THIS^.testStartsWith(
	stringToTest := "",
	expectedString := ""
);
THIS^.testStartsWith(
	stringToTest := "not empty",
	expectedString := ""
);
THIS^.testStartsWith(
	stringToTest := "",
	expectedString := "not empty"
);
THIS^.testStartsWith(
	stringToTest := "not empty",
	expectedString := "not empty"
);
THIS^.testStartsWith(
	stringToTest := "{|}~",
	expectedString := "3649213469328"
);
THIS^.testStartsWith(
	stringToTest := "1one!",
	expectedString := "1"
);
THIS^.testStartsWith(
	stringToTest := "1one!",
	expectedString := "one"
);
THIS^.testStartsWith(
	stringToTest := "1one!",
	expectedString := "!"
);
THIS^.testStartsWith(
	stringToTest := "$0040$n$t$$$"$"",
	expectedString := "$n$t"
);
THIS^.testStartsWith(
	stringToTest := "$n$t$0040$$$"$"",
	expectedString := "$n$t"
);
THIS^.testStartsWith(
	stringToTest := "frontmiddleback",
	expectedString := "front"
);
THIS^.testStartsWith(
	stringToTest := "frontmiddleback",
	expectedString := "frontmiddlebackfront"
);
THIS^.testStartsWith(
	stringToTest := "backfrontmiddle",
	expectedString := "backmiddle"
);
THIS^.testStartsWith(
	stringToTest := "J;%_iTxQSk?6GfWewt}yMKh1)VXqPA@P1YQ:{EAg:8VJ,/FM;j)xJ[[AvYp/}}SzEgtfYS,1K0.5VtA+VJrB(p#55h2z##mw#F)Y@P6Jz9G@6vb=x#E!cYk(Svr@S*KiPJr1VZ6AjrNback4G=vBJd.E:=,k3!wmuGDe#ZKMD#Vx%?M_0&L0#vT]J,+)ZvU{w%8X0=:XzthmT0VG0QrwpXXCWpFxu6[b!c.BunYYfLQi.,?ut?-{jrC1phTHL)y",
	expectedString := "J;%_iTxQSk?6GfWewt}yMKh1)VXqPA@P1YQ:{EAg:8VJ,/FM;j)xJ[[AvYp/}}SzEgtfYS,1K0.5VtA+VJrB(p#55h2z##mw#F)Y@P6Jz9G@6vb=x#E!cYk(Svr@S*KiPJr1VZ6AjrNback4G=vBJd.E:=,k3!wmuGDe#ZKMD#Vx%?M_0&L0#vT]J,+)ZvU{w%8X0=:XzthmT0VG0QrwpXXCWpFxu6[b!c.BunYYfLQi.,?ut?-{jrC1phTHL)y"
);
THIS^.testStartsWith(
	stringToTest := "J;%_iTxQSk?6GfWewt}yMKh1)VXqPA@P1YQ:{EAg:8VJ,/FM;j)xJ[[AvYp/}}SzEgtfYS,1K0.5VtA+VJrB(p#55h2z##mw#F)Y@P6Jz9G@6vb=x#E!cYk(Svr@S*KiPJr1VZ6AjrNback4G=vBJd.E:=,k3!wmuGDe#ZKMD#Vx%?M_0&L0#vT]J,+)ZvU{w%8X0=:XzthmT0VG0QrwpXXCWpFxu6[b!c.BunYYfLQi.,?ut?-{jrC1phTHL)y",
	expectedString := "J;%_iTxQSk?6GfWewt}yMKh1)VXqPA@P1YQ:{EAg:8VJ,/FM;j)xJ[[AvYp/}}SzEgtfYS,1K0.5VtA+VJrB(p#55h2z##mw#F)Y@P6Jz9G@6vb=x#E!cYk(Svr@S*KiPJr1VZ6AjrNback4G=vBJd.E:=,k3!wmuGDe#ZKMD#Vx%?M_0&L0#vT]J,+)ZvU{w%8X0=:XzthmT0VG0QrwpXXCWpFxu6[b!c.BunYYfLQi.,?ut?-{jrC1phTHL)x"
);
THIS^.testStartsWith(
	stringToTest := "∮ E⋅da = Q,  n → ∞, ∑ f(i) = ∏ g(i), ∀x∈ℝ: ⌈x⌉ = −⌊−x⌋, α ∧ ¬β = ¬(¬α ∨ β)",
	expectedString := "∮ E⋅da = Q,  n → ∞"
);
THIS^.testStartsWith(
	stringToTest := "ℕ ⊆ ℕ₀ ⊂ ℤ ⊂ ℚ ⊂ ℝ ⊂ ℂ, ⊥ < a ≠ b ≡ c ≤ d ≪ ⊤ ⇒ (A ⇔ B), 2H₂ + O₂ ⇌ 2H₂O, R = 4.7 kΩ, ⌀ 200 mm",
	expectedString := "ℕ ⊆ ℕ₀ ⊂ ⊂ ℚ ⊂ ℝ ⊂ ℂ"
);
THIS^.testStartsWith(
	stringToTest := "ℕ ⊆ ℕ₀ ⊂ ℤ ⊂ ℚ ⊂ ℝ ⊂ ℂ, ⊥ < a ≠ b ≡ c ≤ d ≪ ⊤ ⇒ (A ⇔ B), 2H₂ + O₂ ⇌ 2H₂O, R = 4.7 kΩ, ⌀ 200 mm",
	expectedString := "ℕ ⊆ ℕ₀ ⊂ ℤ ⊂ ℚ ⊂ ℝ ⊂ ℂ, R = 4.7 kΩ, ⌀ 200 mm"
);
THIS^.testStartsWith(
	stringToTest := "ℕ ⊆ ℕ₀ ⊂ ℤ ⊂ ℚ ⊂ ℝ ⊂ ℂ, ⊥ < a ≠ b ≡ c ≤ d ≪ ⊤ ⇒ (A ⇔ B), 2H₂ + O₂ ⇌ 2H₂O, R = 4.7 kΩ, ⌀ 200 mm",
	expectedString := "ℕ ⊆ ℕ₀ ⊂ ℤ ⊂ ℚ ⊂ ℝ ⊂ ⊥"
);
THIS^.testStartsWith(
	stringToTest := "ði ıntəˈnæʃənəl fəˈnɛtık əsoʊsiˈeıʃn Y [ˈʏpsilɔn], Yen [jɛn], Yoga [ˈjoːgɑ]ˈnæʃənəl fəˈnɛtık ",
	expectedString := "ði ıntəˈnæʃənəl fəˈnɛtık"
);
THIS^.testStartsWith(
	stringToTest := "‚‘„“‘’“We’ve been here”´` †, ‡, ‰, •, 3–4, —, −5/+5, ™, …, 1lI|, 0OD, 8B, €",
	expectedString := "‚‘„“‘’“We’ve been here”´` †, ‡, ‰, •, 3–4, —, −5/+5, ™, …, 1lI|, 0OD, 8B, €"
);
THIS^.testStartsWith(
	stringToTest := "Σὲ γνωρίζω ἀπὸ τὴν κόψη τοῦ σπαθιοῦ τὴν τρομερή,",
	expectedString := "τὴν κόψη τοῦ σπαθ"
);
THIS^.testStartsWith(
	stringToTest := "გთხოვთ ახლავე გაიაროთ რეგისტრაცია Unicode-ის მეათე საერთაშორისო კონფერენციაზე დასასწრებად, რომელიც გაიმართება",
	expectedString := "გთხოვთ ახლავე გაიაროთ რეგისტრაცია"
);
THIS^.testStartsWith(
	stringToTest := "Зарегистрируйтесь сейчас на Десятую Международную Конференцию по Unicode, которая состоится 10-12 марта 1997 года в",
	expectedString := "Международную Конференцию по Unicode, которая"
);
THIS^.testStartsWith(
	stringToTest := "๏ แผ่นดินฮั่นเสื่อมโทรมแสนสังเวช  พระปกเกศกองบู๊กู้ขึ้นใหม่
  สิบสองกษัตริย์ก่อนหน้าแลถัดไป       สององค์ไซร้โง่เขลาเบาปัญญา ",
	expectedString := "๏ แผ่นดินฮั่นเสื่อมโทรมแสนสังเวช " 
);
THIS^.testStartsWith(
	stringToTest := " ሰማይ አይታረስ ንጉሥ አይከሰስ። ብላ ካለኝ እንደአባቴ በቆመጠኝ።",
	expectedString := "አይታረስ ንጉሥ አይከሰስ። በቆመጠኝ።"
);
THIS^.testStartsWith(
	stringToTest := " ᚻᛖ ᚳᚹᚫᚦ ᚦᚫᛏ ᚻᛖ ᛒᚢᛞᛖ ᚩᚾ ᚦᚫᛗ ᛚᚪᚾᛞᛖ ᚾᚩᚱᚦᚹᛖᚪᚱᛞᚢᛗ ᚹᛁᚦ ᚦᚪ ᚹᛖᛥᚫ",
	expectedString := " ᚻᛖ ᚳᚹᚫᚦ ᚦᚫᛏ ᚻᛖ"
);
THIS^.testStartsWith(
	stringToTest := "⡍⠔⠙⠖ ⡊ ⠙⠕⠝⠰⠞ ⠍⠑⠁⠝ ⠞⠕ ⠎⠁⠹ ⠹⠁⠞ ⡊ ⠅⠝⠪⠂ ⠕⠋ ⠍⠹
  ⠪⠝ ⠅⠝⠪⠇⠫⠛⠑⠂ ⠱⠁⠞ ⠹⠻⠑ ⠊⠎ ⠏⠜⠞⠊⠊⠥⠇⠜⠇⠹ ⠙⠑⠁⠙ ⠁⠃⠳⠞",
	expectedString := "⠱⠁⠞ ⠹⠻⠑ ⠊⠎ ⠏⠜⠞⠊⠊⠥⠇⠜⠇⠹ ⠙"
);
THIS^.testStartsWith(
	stringToTest := "╔══╦══╗  ┌──┬──┐  ╭──┬──╮  ╭──┬──╮  ┏━━┳━━┓  ┎┒┏┑   ╷  ╻ ┏┯┓ ┌┰┐    ▊ ╱╲╱╲╳╳╳",
	expectedString := "╔══╦══╗  ┌──┬──┐"
);

THIS^.testStartsWithIgnoreCase(
	stringToTest := "UPPERCASE",
	expectedString := "UPPER"
);
THIS^.testStartsWithIgnoreCase(
	stringToTest := "lowercase",
	expectedString := "lower"
);
THIS^.testStartsWithIgnoreCase(
	stringToTest := "UPPERCASE",
	expectedString := "upper"
);
THIS^.testStartsWithIgnoreCase(
	stringToTest := "lowercase",
	expectedString := "LOWER"
);
THIS^.testStartsWithIgnoreCase(
	stringToTest := "lower",
	expectedString := "UPPER"
);
THIS^.testStartsWithIgnoreCase(
	stringToTest := "⌷←⍳→⍴∆∇⊃‾⍎⍕⌈UPPERCASE",
	expectedString := "⌷←⍳→⍴∆∇⊃‾⍎⍕⌈upper"
);
THIS^.testStartsWithIgnoreCase(
	stringToTest := "⌷←⍳→⍴∆∇⊃‾⍎⍕⌈UPPERCASE",
	expectedString := "⌷←⍳→⍴∆∇⊃‾⍎⍕⌈|upper"
);

THIS^.testStartsWithTrim(
	stringToTest := "$tfrontmiddleback",
	expectedString := "front"
);
THIS^.testStartsWithTrim(
	stringToTest := "frontmiddleback",
	expectedString := "$tfront"
);
THIS^.testStartsWithTrim(
	stringToTest := "$0020frontmiddleback",
	expectedString := "front"
);
THIS^.testStartsWithTrim(
	stringToTest := "frontmiddleback",
	expectedString := "$0020front"
);
THIS^.testStartsWithTrim(
	stringToTest := "$t$n$r$p$lfrontmiddleback",
	expectedString := "$0020$r$t$n$l$pfront"
);
THIS^.testStartsWithTrim(
	stringToTest := "$t$n$r$p$lfrontmiddleback",
	expectedString := "$0020$t$n$r$p$lfront"
);
THIS^.testStartsWithTrim(
	stringToTest := "$t$n$r$p$l⌷←⍳→⍴∆∇⊃‾⍎⍕⌈frontmiddleback$t$n$r$p$l",
	expectedString := "⌷←⍳→⍴∆∇⊃‾⍎⍕⌈front"
);
THIS^.testStartsWithTrim(
	stringToTest := "$t$n$r$p$l⌷←⍳→⍴∆∇⊃‾⍎⍕⌈frontmiddleback$t$n$r$p$l",
	expectedString := "⌷←⍳→⍴∆∇⊃‾⍎⍕front⌈"
);

TcUnit.TEST_FINISHED();
END_METHOD

(*
short summary
==================
This test method tests ``assert.string.unicode.contains``
method of CNM_AssertionInterfaces library with various inputs

.. <legal notes>

legal notes
=================
| SPDX-FileCopyrightText: © 2022 ekvip automation GmbH <info@ekvip.de>
| SPDX-License-Identifier: Apache-2.0
| For details check: Apache-2.0_

.. _Apache-2.0: https://www.apache.org/licenses/LICENSE-2.0

.. </legal notes>

*)


METHOD testContains : BOOL
VAR_INPUT
	(* for the test it's the parameter ``stringToCheck`` *)
	stringToTest 					:WSTRING(Tc2_System.MAX_STRING_LENGTH);
	(* for the test it's the parameter ``searchString`` *)
	expectedString					:WSTRING(Tc2_System.MAX_STRING_LENGTH);
END_VAR
VAR 
	(* just the expectation if the assertion to test must be worng or true *)
	assertionIsWrong				:BOOL;
	(* contains the format string for the test message *)
	message							:Tc2_System.T_MaxString;
	(* used for placeholder string if stringToTest can't be printed *)
	stringToTestAsString 			:Tc2_System.T_MaxString;
	(* used for placeholder string if expectedString can't be printed *)
	expectedStringAsString 			:Tc2_System.T_MaxString;
	(* contains stringToTest in normalized form *)
	normalizedStringToTest			:WSTRING(Tc2_System.MAX_STRING_LENGTH);
	(* contains expectedString in normalized form *)
	normalizedExpectedString		:WSTRING(Tc2_System.MAX_STRING_LENGTH);
	(* holds characterCount of ``expectedString`` *)
	expectedCharacterCount			:UDINT;
	(* TwinCAT printf with the test message *)
	messageStringBuilder			:Tc2_Utilities.FB_FormatString;
	(* hold stringToCheck before assertion *)
	stringToTestBeforeAssertion		:WSTRING(Tc2_System.MAX_STRING_LENGTH);
	(* hold stringToCheck before assertion *)
	expectedStringBeforeAssertion	:WSTRING(Tc2_System.MAX_STRING_LENGTH);
END_VAR
THIS^.assertorContainer.resetAssertor();

stringToTestBeforeAssertion := stringToTest;
expectedStringBeforeAssertion := expectedString;

CNM_UnicodeUtilities.GetUtf16StringLength(
	utf16StringAddress := ADR(expectedString),
	characterCount => expectedCharacterCount
);
assertionIsWrong := ((
		CNM_UnicodeUtilities.FindInUtf16String(
			ADR(stringToTest),
			ADR(expectedString),
		) = 0
	) AND (
		expectedCharacterCount <> 0
	)
);

message := SEL(
	assertionIsWrong,
	'stringToCheck is $'%s$' searchString is $'%s$' assertion must be TRUE', 
	'stringToCheck is $'%s$' searchString is $'%s$' assertion must be FALSE'
);
Tc2_Utilities.WSTRING_TO_STRING2(ADR(stringToTestAsString), ADR(stringToTest), SIZEOF(stringToTestAsString));
Tc2_Utilities.WSTRING_TO_STRING2(ADR(expectedStringAsString), ADR(expectedString), SIZEOF(expectedStringAsString));

IF (
		Tc2_Standard.WLEN(stringToTest) = TO_UINT(Tc2_System.MAX_STRING_LENGTH)
) THEN
	stringToTestAsString := 'String with Tc2_System.MAX_STRING_LENGTH characters';
END_IF
IF (
		Tc2_Standard.WLEN(expectedString) = TO_UINT(Tc2_System.MAX_STRING_LENGTH)
) THEN
	expectedStringAsString := 'String with Tc2_System.MAX_STRING_LENGTH characters';
END_IF

messageStringBuilder(
	sFormat := message,
	arg1 := THIS^.AnyToArg(stringToTestAsString),
	arg2 := THIS^.AnyToArg(expectedStringAsString)
);

THIS^.assertorContainer.assertor.assert.strings.unicode.contains(
	stringToCheck := stringToTest,
	searchString := expectedString,
	ignoreCases := FALSE,
	normalizeStrings := FALSE,
	message			:= ''
);

THIS^.AssertEquals_BOOL(
	Expected 	:= assertionIsWrong,
	Actual 		:= THIS^.assertorContainer.wasAssertionWrong,
	Message 	:= messageStringBuilder.sOut
);

THIS^.AssertEquals_WSTRING(
	Expected 	:= stringToTestBeforeAssertion,
	Actual 		:= stringToTest,
	Message 	:= 'the assertion changed $'stringToTest$''
);

THIS^.AssertEquals_WSTRING(
	Expected 	:= expectedStringBeforeAssertion,
	Actual 		:= expectedString,
	Message 	:= 'the assertion changed $'expectedString$''
);

THIS^.assertorContainer.resetAssertor();

CNM_UnicodeUtilities.NormalizeUtf16String(
	utf16StringBuffer := ADR(stringToTest),
	bufferSize := Tc2_System.MAX_STRING_LENGTH * 2 + 2,
	normalizedStringBuffer := ADR(normalizedStringToTest),
	normalForm := CNM_UnicodeUtilities.NormalizationForm.NFD
);
CNM_UnicodeUtilities.NormalizeUtf16String(
	utf16StringBuffer := ADR(expectedString),
	bufferSize := Tc2_System.MAX_STRING_LENGTH * 2 + 2,
	normalizedStringBuffer := ADR(normalizedExpectedString),
	normalForm := CNM_UnicodeUtilities.NormalizationForm.NFD
);

CNM_UnicodeUtilities.GetUtf16StringLength(
	utf16StringAddress := ADR(normalizedExpectedString),
	characterCount => expectedCharacterCount
);
assertionIsWrong := ((
		CNM_UnicodeUtilities.FindInUtf16String(
			ADR(normalizedStringToTest),
			ADR(normalizedExpectedString),
		) = 0
	) AND (
		expectedCharacterCount <> 0
	)
);

THIS^.assertorContainer.assertor.assert.strings.unicode.contains(
	stringToCheck := stringToTest,
	searchString := expectedString,
	ignoreCases := FALSE,
	normalizeStrings := TRUE,
	message			:= ''
);

THIS^.AssertEquals_BOOL(
	Expected 	:= assertionIsWrong,
	Actual 		:= THIS^.assertorContainer.wasAssertionWrong,
	Message 	:= messageStringBuilder.sOut
);

THIS^.AssertEquals_WSTRING(
	Expected 	:= stringToTestBeforeAssertion,
	Actual 		:= stringToTest,
	Message 	:= 'the assertion changed $'stringToTest$''
);

THIS^.AssertEquals_WSTRING(
	Expected 	:= expectedStringBeforeAssertion,
	Actual 		:= expectedString,
	Message 	:= 'the assertion changed $'expectedString$''
);
END_METHOD

(*
short summary
==================
This test method tests ``assert.string.unicode.contains``
method of CNM_AssertionInterfaces library with various inputs

.. <legal notes>

legal notes
=================
| SPDX-FileCopyrightText: © 2022 ekvip automation GmbH <info@ekvip.de>
| SPDX-License-Identifier: Apache-2.0
| For details check: Apache-2.0_

.. _Apache-2.0: https://www.apache.org/licenses/LICENSE-2.0

.. </legal notes>

*)


METHOD testContainsIgnoreCase : BOOL
VAR_INPUT
	(* for the test it's the parameter ``stringToCheck`` *)
	stringToTest  	:WSTRING(Tc2_System.MAX_STRING_LENGTH);
	(* for the test it's the parameter ``searchString`` *)
	expectedString	:WSTRING(Tc2_System.MAX_STRING_LENGTH);
END_VAR
VAR 
	(* just the expectation if the assertion to test must be worng or true *)
	assertionIsWrong				:BOOL;
	(* contains the format string for the test message *)
	message							:Tc2_System.T_MaxString;
	(* contains ´´stringToTest´´ in upper case *)
	upperStringToTest				:WSTRING(Tc2_System.MAX_STRING_LENGTH);
	(* contains ´´expectedString´´ in upper case *)
	upperExpectedString				:WSTRING(Tc2_System.MAX_STRING_LENGTH);
	(* used for placeholder string if stringToTest can't be printed *)
	stringToTestAsString 			:Tc2_System.T_MaxString;
	(* used for placeholder string if expectedString can't be printed *)
	expectedStringAsString			:Tc2_System.T_MaxString;
	(* contains stringToTest in normalized form *)
	normalizedStringToTest			:WSTRING(Tc2_System.MAX_STRING_LENGTH);
	(* contains expectedString in normalized form *)
	normalizedExpectedString		:WSTRING(Tc2_System.MAX_STRING_LENGTH);
	(* contains stringToTest in normalized form in upper case*)
	normalizedUpperStringToTest		:WSTRING(Tc2_System.MAX_STRING_LENGTH);
	(* contains expectedString in normalized form in upper case*)
	normalizedUpperExpectedString	:WSTRING(Tc2_System.MAX_STRING_LENGTH);
	(* holds characterCount of ``expectedString`` *)
	expectedCharacterCount			:UDINT;
	(* TwinCAT printf with the test message *)
	messageStringBuilder			:Tc2_Utilities.FB_FormatString;
	(* hold stringToCheck before assertion *)
	stringToTestBeforeAssertion		:WSTRING(Tc2_System.MAX_STRING_LENGTH);
	(* hold stringToCheck before assertion *)
	expectedStringBeforeAssertion	:WSTRING(Tc2_System.MAX_STRING_LENGTH);
END_VAR
THIS^.assertorContainer.resetAssertor();

stringToTestBeforeAssertion := stringToTest;
expectedStringBeforeAssertion := expectedString;

upperStringToTest := stringToTest;
upperExpectedString := expectedString;

// both Strings to upper case
CNM_UnicodeUtilities.GetUpperCaseUtf16(ADR(upperStringToTest));
CNM_UnicodeUtilities.GetUpperCaseUtf16(ADR(upperExpectedString));

CNM_UnicodeUtilities.GetUtf16StringLength(
	utf16StringAddress := ADR(upperExpectedString),
	characterCount => expectedCharacterCount
);
assertionIsWrong := ((
		CNM_UnicodeUtilities.FindInUtf16String(
			ADR(upperStringToTest),
			ADR(upperExpectedString),
		) = 0
	) AND (
		expectedCharacterCount <> 0
	)
);

message := SEL(
	assertionIsWrong,
	'stringToCheck is $'%s$' searchString is $'%s$' assertion must be TRUE', 
	'stringToCheck is $'%s$' searchString is $'%s$' assertion must be FALSE'
);

Tc2_Utilities.WSTRING_TO_STRING2(ADR(stringToTestAsString), ADR(stringToTest), SIZEOF(stringToTestAsString));
Tc2_Utilities.WSTRING_TO_STRING2(ADR(expectedStringAsString), ADR(expectedString), SIZEOF(expectedStringAsString));

IF (
		Tc2_Standard.WLEN(stringToTest) = TO_UINT(Tc2_System.MAX_STRING_LENGTH)
) THEN
	stringToTestAsString := 'String with Tc2_System.MAX_STRING_LENGTH characters';
END_IF
IF (
		Tc2_Standard.WLEN(expectedString) = TO_UINT(Tc2_System.MAX_STRING_LENGTH)
) THEN
	expectedStringAsString := 'String with Tc2_System.MAX_STRING_LENGTH characters';
END_IF

messageStringBuilder(
	sFormat := message,
	arg1 := THIS^.AnyToArg(stringToTestAsString),
	arg2 := THIS^.AnyToArg(expectedStringAsString)
);


THIS^.assertorContainer.assertor.assert.strings.unicode.contains(
	stringToCheck := stringToTest,
	searchString := expectedString,
	ignoreCases := TRUE,
	normalizeStrings := FALSE,
	message			:= ''
);

THIS^.AssertEquals_BOOL(
	Expected 	:= assertionIsWrong,
	Actual 		:= THIS^.assertorContainer.wasAssertionWrong,
	Message 	:= messageStringBuilder.sOut
);

THIS^.AssertEquals_WSTRING(
	Expected 	:= stringToTestBeforeAssertion,
	Actual 		:= stringToTest,
	Message 	:= 'the assertion changed $'stringToTest$''
);

THIS^.AssertEquals_WSTRING(
	Expected 	:= expectedStringBeforeAssertion,
	Actual 		:= expectedString,
	Message 	:= 'the assertion changed $'expectedString$''
);

THIS^.assertorContainer.resetAssertor();

CNM_UnicodeUtilities.NormalizeUtf16String(
	utf16StringBuffer := ADR(stringToTest),
	bufferSize := Tc2_System.MAX_STRING_LENGTH * 2 + 2,
	normalizedStringBuffer := ADR(normalizedStringToTest),
	normalForm := CNM_UnicodeUtilities.NormalizationForm.NFD
);
CNM_UnicodeUtilities.NormalizeUtf16String(
	utf16StringBuffer := ADR(expectedString),
	bufferSize := Tc2_System.MAX_STRING_LENGTH * 2 + 2,
	normalizedStringBuffer := ADR(normalizedExpectedString),
	normalForm := CNM_UnicodeUtilities.NormalizationForm.NFD
);

normalizedUpperStringToTest := normalizedStringToTest;
normalizedUpperExpectedString := normalizedExpectedString;
CNM_UnicodeUtilities.GetUpperCaseUtf16(ADR(normalizedUpperStringToTest));
CNM_UnicodeUtilities.GetUpperCaseUtf16(ADR(normalizedUpperExpectedString));


CNM_UnicodeUtilities.GetUtf16StringLength(
	utf16StringAddress := ADR(normalizedUpperExpectedString),
	characterCount => expectedCharacterCount
);
assertionIsWrong := ((
		CNM_UnicodeUtilities.FindInUtf16String(
			ADR(normalizedUpperStringToTest),
			ADR(normalizedUpperExpectedString),
		) = 0
	) AND (
		expectedCharacterCount <> 0
	)
);

THIS^.assertorContainer.assertor.assert.strings.unicode.contains(
	stringToCheck := stringToTest,
	searchString := expectedString,
	ignoreCases := TRUE,
	normalizeStrings := TRUE,
	message			:= ''
);

THIS^.AssertEquals_BOOL(
	Expected 	:= assertionIsWrong,
	Actual 		:= THIS^.assertorContainer.wasAssertionWrong,
	Message 	:= messageStringBuilder.sOut
);

THIS^.AssertEquals_WSTRING(
	Expected 	:= stringToTestBeforeAssertion,
	Actual 		:= stringToTest,
	Message 	:= 'the assertion changed $'stringToTest$''
);

THIS^.AssertEquals_WSTRING(
	Expected 	:= expectedStringBeforeAssertion,
	Actual 		:= expectedString,
	Message 	:= 'the assertion changed $'expectedString$''
);
END_METHOD

(*
short summary
==================
This test method tests ``assert.string.unicode.containsNo``
method of CNM_AssertionInterfaces library with various inputs

.. <legal notes>

legal notes
=================
| SPDX-FileCopyrightText: © 2022 ekvip automation GmbH <info@ekvip.de>
| SPDX-License-Identifier: Apache-2.0
| For details check: Apache-2.0_

.. _Apache-2.0: https://www.apache.org/licenses/LICENSE-2.0

.. </legal notes>

*)


METHOD testContainsNo : BOOL
VAR_INPUT
	(* for the test it's the parameter ``stringToCheck`` *)
	stringToTest  			:WSTRING(Tc2_System.MAX_STRING_LENGTH);
	(* for the test it's the parameter ``searchString`` *)
	expectedString			:WSTRING(Tc2_System.MAX_STRING_LENGTH);
END_VAR
VAR 
	(* just the expectation if the assertion to test must be worng or true *)
	assertionIsWrong				:BOOL;
	(* contains the format string for the test message *)
	message							:Tc2_System.T_MaxString;
	(* used for placeholder string if stringToTest can't be printed *)
	stringToTestAsString 			:Tc2_System.T_MaxString;
	(* used for placeholder string if expectedString can't be printed *)
	expectedStringAsString 			:Tc2_System.T_MaxString;
	(* contains stringToTest in normalized form *)
	normalizedStringToTest			:WSTRING(Tc2_System.MAX_STRING_LENGTH);
	(* contains expectedString in normalized form *)
	normalizedExpectedString		:WSTRING(Tc2_System.MAX_STRING_LENGTH);
	(* holds characterCount of ``expectedString`` *)
	expectedCharacterCount			:UDINT;
	(* TwinCAT printf with the test message *)
	messageStringBuilder			:Tc2_Utilities.FB_FormatString;
	(* hold stringToCheck before assertion *)
	stringToTestBeforeAssertion		:WSTRING(Tc2_System.MAX_STRING_LENGTH);
	(* hold stringToCheck before assertion *)
	expectedStringBeforeAssertion	:WSTRING(Tc2_System.MAX_STRING_LENGTH);
END_VAR
THIS^.assertorContainer.resetAssertor();

stringToTestBeforeAssertion := stringToTest;
expectedStringBeforeAssertion := expectedString;

CNM_UnicodeUtilities.GetUtf16StringLength(
	utf16StringAddress := ADR(expectedString),
	characterCount => expectedCharacterCount
);
assertionIsWrong := ((
		CNM_UnicodeUtilities.FindInUtf16String(
			ADR(stringToTest),
			ADR(expectedString),
		) > 0
	) OR (
		expectedCharacterCount = 0
	)
);

message := SEL(
	assertionIsWrong,
	'stringToCheck is $'%s$' searchString is $'%s$' assertion must be TRUE', 
	'stringToCheck is $'%s$' searchString is $'%s$' assertion must be FALSE'
);

Tc2_Utilities.WSTRING_TO_STRING2(ADR(stringToTestAsString), ADR(stringToTest), SIZEOF(stringToTestAsString));
Tc2_Utilities.WSTRING_TO_STRING2(ADR(expectedStringAsString), ADR(expectedString), SIZEOF(expectedStringAsString));

IF (
		Tc2_Standard.WLEN(stringToTest) = TO_UINT(Tc2_System.MAX_STRING_LENGTH)
) THEN
	stringToTestAsString := 'String with Tc2_System.MAX_STRING_LENGTH characters';
END_IF
IF (
		Tc2_Standard.WLEN(expectedString) = TO_UINT(Tc2_System.MAX_STRING_LENGTH)
) THEN
	expectedStringAsString := 'String with Tc2_System.MAX_STRING_LENGTH characters';
END_IF

messageStringBuilder(
	sFormat := message,
	arg1 := THIS^.AnyToArg(stringToTestAsString),
	arg2 := THIS^.AnyToArg(expectedStringAsString)
);


THIS^.assertorContainer.assertor.assert.strings.unicode.containsNo(
	stringToCheck := stringToTest,
	searchString := expectedString,
	ignoreCases := FALSE,
	normalizeStrings := FALSE,
	message			:= ''
);

THIS^.AssertEquals_BOOL(
	Expected 	:= assertionIsWrong,
	Actual 		:= THIS^.assertorContainer.wasAssertionWrong,
	Message 	:= messageStringBuilder.sOut
);

THIS^.AssertEquals_WSTRING(
	Expected 	:= stringToTestBeforeAssertion,
	Actual 		:= stringToTest,
	Message 	:= 'the assertion changed $'stringToTest$''
);

THIS^.AssertEquals_WSTRING(
	Expected 	:= expectedStringBeforeAssertion,
	Actual 		:= expectedString,
	Message 	:= 'the assertion changed $'expectedString$''
);

THIS^.assertorContainer.resetAssertor();

CNM_UnicodeUtilities.NormalizeUtf16String(
	utf16StringBuffer := ADR(stringToTest),
	bufferSize := Tc2_System.MAX_STRING_LENGTH * 2 + 2,
	normalizedStringBuffer := ADR(normalizedStringToTest),
	normalForm := CNM_UnicodeUtilities.NormalizationForm.NFD
);
CNM_UnicodeUtilities.NormalizeUtf16String(
	utf16StringBuffer := ADR(expectedString),
	bufferSize := Tc2_System.MAX_STRING_LENGTH * 2 + 2,
	normalizedStringBuffer := ADR(normalizedExpectedString),
	normalForm := CNM_UnicodeUtilities.NormalizationForm.NFD
);

CNM_UnicodeUtilities.GetUtf16StringLength(
	utf16StringAddress := ADR(normalizedExpectedString),
	characterCount => expectedCharacterCount
);
assertionIsWrong := ((
		CNM_UnicodeUtilities.FindInUtf16String(
			ADR(normalizedStringToTest),
			ADR(normalizedExpectedString),
		) > 0
	) OR (
		expectedCharacterCount = 0
	)
);

THIS^.assertorContainer.assertor.assert.strings.unicode.containsNo(
	stringToCheck := stringToTest,
	searchString := expectedString,
	ignoreCases := FALSE,
	normalizeStrings := TRUE,
	message			:= ''
);

THIS^.AssertEquals_BOOL(
	Expected 	:= assertionIsWrong,
	Actual 		:= THIS^.assertorContainer.wasAssertionWrong,
	Message 	:= messageStringBuilder.sOut
);

THIS^.AssertEquals_WSTRING(
	Expected 	:= stringToTestBeforeAssertion,
	Actual 		:= stringToTest,
	Message 	:= 'the assertion changed $'stringToTest$''
);

THIS^.AssertEquals_WSTRING(
	Expected 	:= expectedStringBeforeAssertion,
	Actual 		:= expectedString,
	Message 	:= 'the assertion changed $'expectedString$''
);
END_METHOD

(*
short summary
==================
This test method tests ``assert.string.unicode.containsNo``
method of CNM_AssertionInterfaces library with various inputs

.. <legal notes>

legal notes
=================
| SPDX-FileCopyrightText: © 2022 ekvip automation GmbH <info@ekvip.de>
| SPDX-License-Identifier: Apache-2.0
| For details check: Apache-2.0_

.. _Apache-2.0: https://www.apache.org/licenses/LICENSE-2.0

.. </legal notes>

*)


METHOD testContainsNoIgnoreCase : BOOL
VAR_INPUT
	(* for the test it's the parameter ``stringToCheck`` *)
	stringToTest  	:WSTRING(Tc2_System.MAX_STRING_LENGTH);
	(* for the test it's the parameter ``searchString`` *)
	expectedString	:WSTRING(Tc2_System.MAX_STRING_LENGTH);
END_VAR
VAR 
	(* just the expectation if the assertion to test must be worng or true *)
	assertionIsWrong				:BOOL;
	(* contains the format string for the test message *)
	message							:Tc2_System.T_MaxString;
	(* contains ´´stringToTest´´ in upper case *)
	upperStringToTest				:WSTRING(Tc2_System.MAX_STRING_LENGTH);
	(* contains ´´expectedString´´ in upper case *)
	upperExpectedString				:WSTRING(Tc2_System.MAX_STRING_LENGTH);
	(* used for placeholder string if stringToTest can't be printed *)
	stringToTestAsString 			:Tc2_System.T_MaxString;
	(* used for placeholder string if expectedString can't be printed *)
	expectedStringAsString 			:Tc2_System.T_MaxString;
	(* contains stringToTest in normalized form *)
	normalizedStringToTest			:WSTRING(Tc2_System.MAX_STRING_LENGTH);
	(* contains expectedString in normalized form *)
	normalizedExpectedString		:WSTRING(Tc2_System.MAX_STRING_LENGTH);
	(* contains stringToTest in normalized form in upper case*)
	normalizedUpperStringToTest		:WSTRING(Tc2_System.MAX_STRING_LENGTH);
	(* contains expectedString in normalized form in upper case*)
	normalizedUpperExpectedString	:WSTRING(Tc2_System.MAX_STRING_LENGTH);
	(* holds characterCount of ``expectedString`` *)
	expectedCharacterCount			:UDINT;
	(* TwinCAT printf with the test message *)
	messageStringBuilder			:Tc2_Utilities.FB_FormatString;
	(* hold stringToCheck before assertion *)
	stringToTestBeforeAssertion		:WSTRING(Tc2_System.MAX_STRING_LENGTH);
	(* hold stringToCheck before assertion *)
	expectedStringBeforeAssertion	:WSTRING(Tc2_System.MAX_STRING_LENGTH);
END_VAR
THIS^.assertorContainer.resetAssertor();

stringToTestBeforeAssertion := stringToTest;
expectedStringBeforeAssertion := expectedString;

upperStringToTest := stringToTest;
upperExpectedString := expectedString;

// both Strings to upper case
CNM_UnicodeUtilities.GetUpperCaseUtf16(ADR(upperStringToTest));
CNM_UnicodeUtilities.GetUpperCaseUtf16(ADR(upperExpectedString));

CNM_UnicodeUtilities.GetUtf16StringLength(
	utf16StringAddress := ADR(upperExpectedString),
	characterCount => expectedCharacterCount
);
assertionIsWrong := ((
		CNM_UnicodeUtilities.FindInUtf16String(
			ADR(upperStringToTest),
			ADR(upperExpectedString),
		) > 0
	) OR (
		expectedCharacterCount = 0
	)
);

message := SEL(
	assertionIsWrong,
	'stringToCheck is $'%s$' searchString is $'%s$' assertion must be TRUE', 
	'stringToCheck is $'%s$' searchString is $'%s$' assertion must be FALSE'
);

Tc2_Utilities.WSTRING_TO_STRING2(ADR(stringToTestAsString), ADR(stringToTest), SIZEOF(stringToTestAsString));
Tc2_Utilities.WSTRING_TO_STRING2(ADR(expectedStringAsString), ADR(expectedString), SIZEOF(expectedStringAsString));

IF (
		Tc2_Standard.WLEN(stringToTest) = TO_UINT(Tc2_System.MAX_STRING_LENGTH)
) THEN
	stringToTestAsString := 'String with Tc2_System.MAX_STRING_LENGTH characters';
END_IF
IF (
		Tc2_Standard.WLEN(expectedString) = TO_UINT(Tc2_System.MAX_STRING_LENGTH)
) THEN
	expectedStringAsString := 'String with Tc2_System.MAX_STRING_LENGTH characters';
END_IF

messageStringBuilder(
	sFormat := message,
	arg1 := THIS^.AnyToArg(stringToTestAsString),
	arg2 := THIS^.AnyToArg(expectedStringAsString)
);


THIS^.assertorContainer.assertor.assert.strings.unicode.containsNo(
	stringToCheck := stringToTest,
	searchString := expectedString,
	ignoreCases := TRUE,
	normalizeStrings := FALSE,
	message			:= ''
);

THIS^.AssertEquals_BOOL(
	Expected 	:= assertionIsWrong,
	Actual 		:= THIS^.assertorContainer.wasAssertionWrong,
	Message 	:= messageStringBuilder.sOut
);

THIS^.AssertEquals_WSTRING(
	Expected 	:= stringToTestBeforeAssertion,
	Actual 		:= stringToTest,
	Message 	:= 'the assertion changed $'stringToTest$''
);

THIS^.AssertEquals_WSTRING(
	Expected 	:= expectedStringBeforeAssertion,
	Actual 		:= expectedString,
	Message 	:= 'the assertion changed $'expectedString$''
);

THIS^.assertorContainer.resetAssertor();

CNM_UnicodeUtilities.NormalizeUtf16String(
	utf16StringBuffer := ADR(stringToTest),
	bufferSize := Tc2_System.MAX_STRING_LENGTH * 2 + 2,
	normalizedStringBuffer := ADR(normalizedStringToTest),
	normalForm := CNM_UnicodeUtilities.NormalizationForm.NFD
);
CNM_UnicodeUtilities.NormalizeUtf16String(
	utf16StringBuffer := ADR(expectedString),
	bufferSize := Tc2_System.MAX_STRING_LENGTH * 2 + 2,
	normalizedStringBuffer := ADR(normalizedExpectedString),
	normalForm := CNM_UnicodeUtilities.NormalizationForm.NFD
);

normalizedUpperStringToTest := normalizedStringToTest;
normalizedUpperExpectedString := normalizedExpectedString;
CNM_UnicodeUtilities.GetUpperCaseUtf16(ADR(normalizedUpperStringToTest));
CNM_UnicodeUtilities.GetUpperCaseUtf16(ADR(normalizedUpperExpectedString));


CNM_UnicodeUtilities.GetUtf16StringLength(
	utf16StringAddress := ADR(normalizedUpperExpectedString),
	characterCount => expectedCharacterCount
);
assertionIsWrong := ((
		CNM_UnicodeUtilities.FindInUtf16String(
			ADR(normalizedUpperStringToTest),
			ADR(normalizedUpperExpectedString),
		) > 0
	) OR (
		expectedCharacterCount = 0
	)
);

THIS^.assertorContainer.assertor.assert.strings.unicode.containsNo(
	stringToCheck := stringToTest,
	searchString := expectedString,
	ignoreCases := TRUE,
	normalizeStrings := TRUE,
	message			:= ''
);

THIS^.AssertEquals_BOOL(
	Expected 	:= assertionIsWrong,
	Actual 		:= THIS^.assertorContainer.wasAssertionWrong,
	Message 	:= messageStringBuilder.sOut
);

THIS^.AssertEquals_WSTRING(
	Expected 	:= stringToTestBeforeAssertion,
	Actual 		:= stringToTest,
	Message 	:= 'the assertion changed $'stringToTest$''
);

THIS^.AssertEquals_WSTRING(
	Expected 	:= expectedStringBeforeAssertion,
	Actual 		:= expectedString,
	Message 	:= 'the assertion changed $'expectedString$''
);
END_METHOD

(*
short summary
==================
This test method tests ``assert.string.unicode.endsWith``
method of CNM_AssertionInterfaces library with various inputs

.. <legal notes>

legal notes
=================
| SPDX-FileCopyrightText: © 2022 ekvip automation GmbH <info@ekvip.de>
| SPDX-License-Identifier: Apache-2.0
| For details check: Apache-2.0_

.. _Apache-2.0: https://www.apache.org/licenses/LICENSE-2.0

.. </legal notes>

*)


METHOD testEndsWith : BOOL
VAR_INPUT
	(* for the test it's the parameter ``stringToCheck`` *)
	stringToTest  	:WSTRING(Tc2_System.MAX_STRING_LENGTH);
	(* for the test it's the parameter ``searchString`` *)
	expectedString	:WSTRING(Tc2_System.MAX_STRING_LENGTH);
END_VAR
VAR 
	(* just the expectation if the assertion to test must be worng or true *)
	assertionIsWrong				:BOOL;
	(* contains the format string for the test message *)
	message							:Tc2_System.T_MaxString;
	(* used for placeholder string if stringToTest can't be printed *)
	stringToTestAsString 			:Tc2_System.T_MaxString;
	(* used for placeholder string if expectedString can't be printed *)
	expectedStringAsString 			:Tc2_System.T_MaxString;
	(* contains stringToTest in normalized form *)
	normalizedStringToTest			:WSTRING(Tc2_System.MAX_STRING_LENGTH);
	(* contains expectedString in normalized form *)
	normalizedExpectedString		:WSTRING(Tc2_System.MAX_STRING_LENGTH);
	(* contains the rigth side of ``stringToCheck`` *)
	rigthOfStringToCheck			:WSTRING(Tc2_System.MAX_STRING_LENGTH);
	(* holds characterCount of ``expectedString`` *)
	expectedCharacterCount			:UDINT;
	(* TwinCAT printf with the test message *)
	messageStringBuilder			:Tc2_Utilities.FB_FormatString;
	(* hold stringToCheck before assertion *)
	stringToTestBeforeAssertion		:WSTRING(Tc2_System.MAX_STRING_LENGTH);
	(* hold stringToCheck before assertion *)
	expectedStringBeforeAssertion	:WSTRING(Tc2_System.MAX_STRING_LENGTH);
END_VAR
THIS^.assertorContainer.resetAssertor();

stringToTestBeforeAssertion := stringToTest;
expectedStringBeforeAssertion := expectedString;

CNM_UnicodeUtilities.GetUtf16StringLength(
	utf16StringAddress := ADR(expectedString),
	characterCount => expectedCharacterCount
);
rigthOfStringToCheck := WRIGHT(stringToTest, TO_INT(expectedCharacterCount));
assertionIsWrong := ((
		CNM_UnicodeUtilities.FindInUtf16String(
			ADR(rigthOfStringToCheck),
			ADR(expectedString),
		) <> 1
	) AND (
		expectedCharacterCount <> 0
	)
);

message := SEL(
	assertionIsWrong,
	'stringToCheck is $'%s$' end is $'%s$' assertion must be TRUE', 
	'stringToCheck is $'%s$' end is $'%s$' assertion must be FALSE'
);

Tc2_Utilities.WSTRING_TO_STRING2(ADR(stringToTestAsString), ADR(stringToTest), SIZEOF(stringToTestAsString));
Tc2_Utilities.WSTRING_TO_STRING2(ADR(expectedStringAsString), ADR(expectedString), SIZEOF(expectedStringAsString));

IF (
		Tc2_Standard.WLEN(stringToTest) = TO_UINT(Tc2_System.MAX_STRING_LENGTH)
) THEN
	stringToTestAsString := 'String with Tc2_System.MAX_STRING_LENGTH characters';
END_IF
IF (
		Tc2_Standard.WLEN(expectedString) = TO_UINT(Tc2_System.MAX_STRING_LENGTH)
) THEN
	expectedStringAsString := 'String with Tc2_System.MAX_STRING_LENGTH characters';
END_IF

messageStringBuilder(
	sFormat := message,
	arg1 := THIS^.AnyToArg(stringToTestAsString),
	arg2 := THIS^.AnyToArg(expectedStringAsString)
);


THIS^.assertorContainer.assertor.assert.strings.unicode.endsWith(
	stringToCheck := stringToTest,
	end := expectedString,
	ignoreCases := FALSE,
	trim := FALSE,
	normalizeStrings := FALSE,
	message			:= ''
);

THIS^.AssertEquals_BOOL(
	Expected 	:= assertionIsWrong,
	Actual 		:= THIS^.assertorContainer.wasAssertionWrong,
	Message 	:= messageStringBuilder.sOut
);

THIS^.AssertEquals_WSTRING(
	Expected 	:= stringToTestBeforeAssertion,
	Actual 		:= stringToTest,
	Message 	:= 'the assertion changed $'stringToTest$''
);

THIS^.AssertEquals_WSTRING(
	Expected 	:= expectedStringBeforeAssertion,
	Actual 		:= expectedString,
	Message 	:= 'the assertion changed $'expectedString$''
);

THIS^.assertorContainer.resetAssertor();

CNM_UnicodeUtilities.NormalizeUtf16String(
	utf16StringBuffer := ADR(stringToTest),
	bufferSize := Tc2_System.MAX_STRING_LENGTH * 2 + 2,
	normalizedStringBuffer := ADR(normalizedStringToTest),
	normalForm := CNM_UnicodeUtilities.NormalizationForm.NFD
);
CNM_UnicodeUtilities.NormalizeUtf16String(
	utf16StringBuffer := ADR(expectedString),
	bufferSize := Tc2_System.MAX_STRING_LENGTH * 2 + 2,
	normalizedStringBuffer := ADR(normalizedExpectedString),
	normalForm := CNM_UnicodeUtilities.NormalizationForm.NFD
);

CNM_UnicodeUtilities.GetUtf16StringLength(
	utf16StringAddress := ADR(normalizedExpectedString),
	characterCount => expectedCharacterCount
);
rigthOfStringToCheck := WRIGHT(normalizedStringToTest, TO_INT(expectedCharacterCount));
assertionIsWrong := ((
		CNM_UnicodeUtilities.FindInUtf16String(
			ADR(rigthOfStringToCheck),
			ADR(normalizedExpectedString),
		) <> 1
	) AND (
		expectedCharacterCount <> 0
	)
);

THIS^.assertorContainer.assertor.assert.strings.unicode.endsWith(
	stringToCheck := stringToTest,
	end := expectedString,
	ignoreCases := FALSE,
	trim		:= FALSE,
	normalizeStrings := TRUE,
	message			:= ''
);

THIS^.AssertEquals_BOOL(
	Expected 	:= assertionIsWrong,
	Actual 		:= THIS^.assertorContainer.wasAssertionWrong,
	Message 	:= messageStringBuilder.sOut
);

THIS^.AssertEquals_WSTRING(
	Expected 	:= stringToTestBeforeAssertion,
	Actual 		:= stringToTest,
	Message 	:= 'the assertion changed $'stringToTest$''
);

THIS^.AssertEquals_WSTRING(
	Expected 	:= expectedStringBeforeAssertion,
	Actual 		:= expectedString,
	Message 	:= 'the assertion changed $'expectedString$''
);
END_METHOD

(*
short summary
==================
This test method tests ``assert.string.unicode.endsWith``
method of CNM_AssertionInterfaces library with various inputs

.. <legal notes>

legal notes
=================
| SPDX-FileCopyrightText: © 2022 ekvip automation GmbH <info@ekvip.de>
| SPDX-License-Identifier: Apache-2.0
| For details check: Apache-2.0_

.. _Apache-2.0: https://www.apache.org/licenses/LICENSE-2.0

.. </legal notes>

*)


METHOD testEndsWithIgnoreCase : BOOL
VAR_INPUT
	(* for the test it's the parameter ``stringToCheck`` *)
	stringToTest  	:WSTRING(Tc2_System.MAX_STRING_LENGTH);
	(* for the test it's the parameter ``searchString`` *)
	expectedString	:WSTRING(Tc2_System.MAX_STRING_LENGTH);
END_VAR
VAR 
	(* just the expectation if the assertion to test must be worng or true *)
	assertionIsWrong				:BOOL;
	(* contains the format string for the test message *)
	message							:Tc2_System.T_MaxString;
	(* contains ´´stringToTest´´ in upper case *)
	upperStringToTest				:WSTRING(Tc2_System.MAX_STRING_LENGTH);
	(* contains ´´expectedString´´ in upper case *)
	upperExpectedString				:WSTRING(Tc2_System.MAX_STRING_LENGTH);
	(* used for placeholder string if stringToTest can't be printed *)
	stringToTestAsString 			:Tc2_System.T_MaxString;
	(* used for placeholder string if expectedString can't be printed *)
	expectedStringAsString 			:Tc2_System.T_MaxString;
	(* contains the rigth side of ``stringToCheck`` *)
	rigthOfStringToCheck			:WSTRING(Tc2_System.MAX_STRING_LENGTH);
	(* contains stringToTest in normalized form *)
	normalizedStringToTest			:WSTRING(Tc2_System.MAX_STRING_LENGTH);
	(* contains expectedString in normalized form *)
	normalizedExpectedString		:WSTRING(Tc2_System.MAX_STRING_LENGTH);
	(* contains stringToTest in normalized form in upper case*)
	normalizedUpperStringToTest		:WSTRING(Tc2_System.MAX_STRING_LENGTH);
	(* contains expectedString in normalized form in upper case*)
	normalizedUpperExpectedString	:WSTRING(Tc2_System.MAX_STRING_LENGTH);
	(* holds characterCount of ``expectedString`` *)
	expectedCharacterCount			:UDINT;
	(* TwinCAT printf with the test message *)
	messageStringBuilder			:Tc2_Utilities.FB_FormatString;
	(* hold stringToCheck before assertion *)
	stringToTestBeforeAssertion		:WSTRING(Tc2_System.MAX_STRING_LENGTH);
	(* hold stringToCheck before assertion *)
	expectedStringBeforeAssertion	:WSTRING(Tc2_System.MAX_STRING_LENGTH);
END_VAR
THIS^.assertorContainer.resetAssertor();

stringToTestBeforeAssertion := stringToTest;
expectedStringBeforeAssertion := expectedString;

upperStringToTest := stringToTest;
upperExpectedString := expectedString;

// both Strings to upper case
CNM_UnicodeUtilities.GetUpperCaseUtf16(ADR(upperStringToTest));
CNM_UnicodeUtilities.GetUpperCaseUtf16(ADR(upperExpectedString));

CNM_UnicodeUtilities.GetUtf16StringLength(
	utf16StringAddress := ADR(upperExpectedString),
	characterCount => expectedCharacterCount
);
rigthOfStringToCheck := WRIGHT(upperStringToTest, TO_INT(expectedCharacterCount));
assertionIsWrong := ((
		CNM_UnicodeUtilities.FindInUtf16String(
			ADR(rigthOfStringToCheck),
			ADR(upperExpectedString),
		) <> 1
	) AND (
		expectedCharacterCount <> 0
	)
);
message := SEL(
	assertionIsWrong,
	'stringToCheck is $'%s$' end is $'%s$' assertion must be TRUE', 
	'stringToCheck is $'%s$' end is $'%s$' assertion must be FALSE'
);

Tc2_Utilities.WSTRING_TO_STRING2(ADR(stringToTestAsString), ADR(stringToTest), SIZEOF(stringToTestAsString));
Tc2_Utilities.WSTRING_TO_STRING2(ADR(expectedStringAsString), ADR(expectedString), SIZEOF(expectedStringAsString));

IF (
		Tc2_Standard.WLEN(stringToTest) = TO_UINT(Tc2_System.MAX_STRING_LENGTH)
) THEN
	stringToTestAsString := 'String with Tc2_System.MAX_STRING_LENGTH characters';
END_IF
IF (
		Tc2_Standard.WLEN(expectedString) = TO_UINT(Tc2_System.MAX_STRING_LENGTH)
) THEN
	expectedStringAsString := 'String with Tc2_System.MAX_STRING_LENGTH characters';
END_IF

messageStringBuilder(
	sFormat := message,
	arg1 := THIS^.AnyToArg(stringToTestAsString),
	arg2 := THIS^.AnyToArg(expectedStringAsString)
);


THIS^.assertorContainer.assertor.assert.strings.unicode.endsWith(
	stringToCheck := stringToTest,
	end := expectedString,
	ignoreCases := TRUE,
	trim := FALSE,
	normalizeStrings := FALSE,
	message			:= ''
);

THIS^.AssertEquals_BOOL(
	Expected 	:= assertionIsWrong,
	Actual 		:= THIS^.assertorContainer.wasAssertionWrong,
	Message 	:= messageStringBuilder.sOut
);

THIS^.AssertEquals_WSTRING(
	Expected 	:= stringToTestBeforeAssertion,
	Actual 		:= stringToTest,
	Message 	:= 'the assertion changed $'stringToTest$''
);

THIS^.AssertEquals_WSTRING(
	Expected 	:= expectedStringBeforeAssertion,
	Actual 		:= expectedString,
	Message 	:= 'the assertion changed $'expectedString$''
);

CNM_UnicodeUtilities.NormalizeUtf16String(
	utf16StringBuffer := ADR(stringToTest),
	bufferSize := Tc2_System.MAX_STRING_LENGTH * 2 + 2,
	normalizedStringBuffer := ADR(normalizedStringToTest),
	normalForm := CNM_UnicodeUtilities.NormalizationForm.NFD
);
CNM_UnicodeUtilities.NormalizeUtf16String(
	utf16StringBuffer := ADR(expectedString),
	bufferSize := Tc2_System.MAX_STRING_LENGTH * 2 + 2,
	normalizedStringBuffer := ADR(normalizedExpectedString),
	normalForm := CNM_UnicodeUtilities.NormalizationForm.NFD
);
THIS^.assertorContainer.resetAssertor();

normalizedUpperStringToTest := normalizedStringToTest;
normalizedUpperExpectedString := normalizedExpectedString;
CNM_UnicodeUtilities.GetUpperCaseUtf16(ADR(normalizedUpperStringToTest));
CNM_UnicodeUtilities.GetUpperCaseUtf16(ADR(normalizedUpperExpectedString));


CNM_UnicodeUtilities.GetUtf16StringLength(
	utf16StringAddress := ADR(normalizedUpperExpectedString),
	characterCount => expectedCharacterCount
);
rigthOfStringToCheck := WRIGHT(normalizedUpperStringToTest, TO_INT(expectedCharacterCount));
assertionIsWrong := ((
		CNM_UnicodeUtilities.FindInUtf16String(
			ADR(rigthOfStringToCheck),
			ADR(normalizedUpperExpectedString),
		) <> 1
	) AND (
		expectedCharacterCount <> 0
	)
);

THIS^.assertorContainer.assertor.assert.strings.unicode.endsWith(
	stringToCheck := stringToTest,
	end := expectedString,
	ignoreCases := TRUE,
	trim		:= FALSE,
	normalizeStrings := TRUE,
	message			:= ''
);

THIS^.AssertEquals_BOOL(
	Expected 	:= assertionIsWrong,
	Actual 		:= THIS^.assertorContainer.wasAssertionWrong,
	Message 	:= messageStringBuilder.sOut
);

THIS^.AssertEquals_WSTRING(
	Expected 	:= stringToTestBeforeAssertion,
	Actual 		:= stringToTest,
	Message 	:= 'the assertion changed $'stringToTest$''
);

THIS^.AssertEquals_WSTRING(
	Expected 	:= expectedStringBeforeAssertion,
	Actual 		:= expectedString,
	Message 	:= 'the assertion changed $'expectedString$''
);
END_METHOD

(*
short summary
==================
This test method tests ``assert.string.unicode.endsWith``
method of CNM_AssertionInterfaces library with various inputs

.. <legal notes>

legal notes
=================
| SPDX-FileCopyrightText: © 2022 ekvip automation GmbH <info@ekvip.de>
| SPDX-License-Identifier: Apache-2.0
| For details check: Apache-2.0_

.. _Apache-2.0: https://www.apache.org/licenses/LICENSE-2.0

.. </legal notes>

*)


METHOD testEndsWithTrim : BOOL
VAR_INPUT
	(* for the test it's the parameter ``stringToCheck`` *)
	stringToTest 	:WSTRING(Tc2_System.MAX_STRING_LENGTH);
	(* for the test it's the parameter ``end`` *)
	expectedString :WSTRING(Tc2_System.MAX_STRING_LENGTH);
END_VAR
VAR 
	(* just the expectation if the assertion to test must be worng or true *)
	assertionIsWrong				:BOOL;
	(* contains the format string for the test message *)
	message							:Tc2_System.T_MaxString;
	(* contains trimed ´´stringToTest´´ *)
	trimedStringToTest				:WSTRING(Tc2_System.MAX_STRING_LENGTH);
	(* contains trimed ´´expectedString´´ *)
	trimedExpectedString			:WSTRING(Tc2_System.MAX_STRING_LENGTH);
	(* used for placeholder string if stringToTest can't be printed *)
	stringToTestAsString	 		:Tc2_System.T_MaxString;
	(* used for placeholder string if expectedString can't be printed *)
	expectedStringAsString 			:Tc2_System.T_MaxString;
	(* right side of ``stringToCheck`` *)
	rigthOfStringToCheck			:WSTRING(Tc2_System.MAX_STRING_LENGTH);
	(* contains stringToTest in normalized form *)
	normalizedStringToTest			:WSTRING(Tc2_System.MAX_STRING_LENGTH);
	(* contains expectedString in normalized form *)
	normalizedExpectedString		:WSTRING(Tc2_System.MAX_STRING_LENGTH);
	(* contains stringToTest in normalized form trimed *)
	normalizedTrimedStringToTest	:WSTRING(Tc2_System.MAX_STRING_LENGTH);
	(* contains expectedString in normalized form trimed *)
	normalizedTrimedExpectedString	:WSTRING(Tc2_System.MAX_STRING_LENGTH);
	(* holds characterCount of ``expectedString`` *)
	expectedCharacterCount			:UDINT;
	(* TwinCAT printf with the test message *)
	messageStringBuilder			:Tc2_Utilities.FB_FormatString;
	(* hold stringToCheck before assertion *)
	stringToTestBeforeAssertion		:WSTRING(Tc2_System.MAX_STRING_LENGTH);
	(* hold stringToCheck before assertion *)
	expectedStringBeforeAssertion	:WSTRING(Tc2_System.MAX_STRING_LENGTH);
END_VAR
THIS^.assertorContainer.resetAssertor();

stringToTestBeforeAssertion := stringToTest;
expectedStringBeforeAssertion := expectedString;

trimedStringToTest := stringToTest;
trimedExpectedString := expectedString;

// trim the right of both strings
CNM_UnicodeUtilities.TrimRightUtf16String(ADR(trimedStringToTest));
CNM_UnicodeUtilities.TrimRightUtf16String(ADR(trimedExpectedString));

CNM_UnicodeUtilities.GetUtf16StringLength(
	utf16StringAddress := ADR(trimedExpectedString),
	characterCount => expectedCharacterCount
);
rigthOfStringToCheck := WRIGHT(trimedStringToTest, TO_INT(expectedCharacterCount));
assertionIsWrong := ((
		CNM_UnicodeUtilities.FindInUtf16String(
			ADR(rigthOfStringToCheck),
			ADR(trimedExpectedString),
		) <> 1
	) AND (
		expectedCharacterCount <> 0
	)
);

message := SEL(
	assertionIsWrong,
	'stringToCheck is $'%s$' end is $'%s$' assertion must be TRUE', 
	'stringToCheck is $'%s$' end is $'%s$' assertion must be FALSE'
);

Tc2_Utilities.WSTRING_TO_STRING2(ADR(stringToTestAsString), ADR(stringToTest), SIZEOF(stringToTestAsString));
Tc2_Utilities.WSTRING_TO_STRING2(ADR(expectedStringAsString), ADR(expectedString), SIZEOF(expectedStringAsString));

IF (
		Tc2_Standard.WLEN(stringToTest) = TO_UINT(Tc2_System.MAX_STRING_LENGTH)
) THEN
	stringToTestAsString := 'String with Tc2_System.MAX_STRING_LENGTH characters';
END_IF
IF (
		Tc2_Standard.WLEN(expectedString) = TO_UINT(Tc2_System.MAX_STRING_LENGTH)
) THEN
	expectedStringAsString := 'String with Tc2_System.MAX_STRING_LENGTH characters';
END_IF

messageStringBuilder(
	sFormat := message,
	arg1 := THIS^.AnyToArg(stringToTestAsString),
	arg2 := THIS^.AnyToArg(expectedStringAsString)
);


THIS^.assertorContainer.assertor.assert.strings.unicode.endsWith(
	stringToCheck := stringToTest,
	end := expectedString,
	ignoreCases := FALSE,
	trim := TRUE,
	normalizeStrings := FALSE,
	message			:= ''
);

THIS^.AssertEquals_BOOL(
	Expected 	:= assertionIsWrong,
	Actual 		:= THIS^.assertorContainer.wasAssertionWrong,
	Message 	:= messageStringBuilder.sOut
);

THIS^.AssertEquals_WSTRING(
	Expected 	:= stringToTestBeforeAssertion,
	Actual 		:= stringToTest,
	Message 	:= 'the assertion changed $'stringToTest$''
);

THIS^.AssertEquals_WSTRING(
	Expected 	:= expectedStringBeforeAssertion,
	Actual 		:= expectedString,
	Message 	:= 'the assertion changed $'expectedString$''
);

THIS^.assertorContainer.resetAssertor();

CNM_UnicodeUtilities.NormalizeUtf16String(
	utf16StringBuffer := ADR(stringToTest),
	bufferSize := Tc2_System.MAX_STRING_LENGTH * 2 + 2,
	normalizedStringBuffer := ADR(normalizedStringToTest),
	normalForm := CNM_UnicodeUtilities.NormalizationForm.NFD
);
CNM_UnicodeUtilities.NormalizeUtf16String(
	utf16StringBuffer := ADR(expectedString),
	bufferSize := Tc2_System.MAX_STRING_LENGTH * 2 + 2,
	normalizedStringBuffer := ADR(normalizedExpectedString),
	normalForm := CNM_UnicodeUtilities.NormalizationForm.NFD
);
THIS^.assertorContainer.resetAssertor();

normalizedTrimedStringToTest := normalizedStringToTest;
normalizedTrimedExpectedString := normalizedExpectedString;
CNM_UnicodeUtilities.TrimRightUtf16String(ADR(normalizedTrimedStringToTest));
CNM_UnicodeUtilities.TrimRightUtf16String(ADR(normalizedTrimedExpectedString));

CNM_UnicodeUtilities.GetUtf16StringLength(
	utf16StringAddress := ADR(normalizedTrimedExpectedString),
	characterCount => expectedCharacterCount
);
rigthOfStringToCheck := WRIGHT(normalizedTrimedStringToTest, TO_INT(expectedCharacterCount));
assertionIsWrong := ((
		CNM_UnicodeUtilities.FindInUtf16String(
			ADR(rigthOfStringToCheck),
			ADR(normalizedTrimedExpectedString),
		) <> 1
	) AND (
		expectedCharacterCount <> 0
	)
);

THIS^.assertorContainer.assertor.assert.strings.unicode.endsWith(
	stringToCheck := stringToTest,
	end := expectedString,
	ignoreCases := FALSE,
	trim		:= TRUE,
	normalizeStrings := TRUE,
	message			:= ''
);

THIS^.AssertEquals_BOOL(
	Expected 	:= assertionIsWrong,
	Actual 		:= THIS^.assertorContainer.wasAssertionWrong,
	Message 	:= messageStringBuilder.sOut
);

THIS^.AssertEquals_WSTRING(
	Expected 	:= stringToTestBeforeAssertion,
	Actual 		:= stringToTest,
	Message 	:= 'the assertion changed $'stringToTest$''
);

THIS^.AssertEquals_WSTRING(
	Expected 	:= expectedStringBeforeAssertion,
	Actual 		:= expectedString,
	Message 	:= 'the assertion changed $'expectedString$''
);
END_METHOD

(*
short summary
==================
This test method tests ``assert.string.unicode.isEmpty``
method of CNM_AssertionInterfaces library with various inputs

.. <legal notes>

legal notes
=================
| SPDX-FileCopyrightText: © 2022 ekvip automation GmbH <info@ekvip.de>
| SPDX-License-Identifier: Apache-2.0
| For details check: Apache-2.0_

.. _Apache-2.0: https://www.apache.org/licenses/LICENSE-2.0

.. </legal notes>

*)


METHOD testisEmpty : BOOL
VAR_INPUT
	(* for the test it's the parameter ``stringToCheck`` *)
	stringToTest :WSTRING(Tc2_System.MAX_STRING_LENGTH);
END_VAR
VAR 
	(* just the expectation if the assertion to test must be worng or true *)
	assertionIsWrong				:BOOL;
	(* contains the format string for the test message *)
	message							:Tc2_System.T_MaxString;
	(* used for placeholder string if stringToTest can't be printed *)
	stringToTestAsString 			:Tc2_System.T_MaxString;
	(* holds characterCount of ``stringToTest`` *)
	stringToTestCharacterCount		:UDINT;
	(* TwinCAT printf with the test message *)
	messageStringBuilder			:Tc2_Utilities.FB_FormatString;
	(* hold stringToCheck before assertion *)
	stringToTestBeforeAssertion		:WSTRING(Tc2_System.MAX_STRING_LENGTH);
END_VAR
THIS^.assertorContainer.resetAssertor();

stringToTestBeforeAssertion := stringToTest;

CNM_UnicodeUtilities.GetUtf16StringLength(
	utf16StringAddress := ADR(stringToTest),
	characterCount => stringToTestCharacterCount
);
assertionIsWrong :=  stringToTestCharacterCount > 0;

message := SEL(
	assertionIsWrong,
	'stringToCheck is $'%s$' assertion must be TRUE', 
	'stringToCheck is $'%s$' assertion must be FALSE'
);

Tc2_Utilities.WSTRING_TO_STRING2(ADR(stringToTestAsString), ADR(stringToTest), SIZEOF(stringToTestAsString));

IF (
		Tc2_Standard.WLEN(stringToTest) = TO_UINT(Tc2_System.MAX_STRING_LENGTH)
) THEN
	stringToTestAsString := 'String with Tc2_System.MAX_STRING_LENGTH characters';
END_IF

messageStringBuilder(
	sFormat := message,
	arg1 := THIS^.AnyToArg(stringToTestAsString),
);


THIS^.assertorContainer.assertor.assert.strings.unicode.isEmpty(
	stringToCheck := stringToTest,
	message			:= ''
);

THIS^.AssertEquals_BOOL(
	Expected 	:= assertionIsWrong,
	Actual 		:= THIS^.assertorContainer.wasAssertionWrong,
	Message 	:= messageStringBuilder.sOut
);

THIS^.AssertEquals_WSTRING(
	Expected 	:= stringToTestBeforeAssertion,
	Actual 		:= stringToTest,
	Message 	:= 'the assertion changed $'stringToTest$''
);
END_METHOD

(*
short summary
==================
This test method tests ``assert.string.unicode.isEqualTo``
method of CNM_AssertionInterfaces library with various inputs

.. <legal notes>

legal notes
=================
| SPDX-FileCopyrightText: © 2022 ekvip automation GmbH <info@ekvip.de>
| SPDX-License-Identifier: Apache-2.0
| For details check: Apache-2.0_

.. _Apache-2.0: https://www.apache.org/licenses/LICENSE-2.0

.. </legal notes>

*)


METHOD testIsEqualTo : BOOL
VAR_INPUT
	(* for the test it's the parameter ``stringToCheck`` *)
	stringToTest  	:WSTRING(Tc2_System.MAX_STRING_LENGTH);
	(* for the test it's the parameter ``searchString`` *)
	expectedString	:WSTRING(Tc2_System.MAX_STRING_LENGTH);
END_VAR
VAR 
	(* just the expectation if the assertion to test must be worng or true *)
	assertionIsWrong				:BOOL;
	(* contains the format string for the test message *)
	message							:Tc2_System.T_MaxString;
	(* used for placeholder string if stringToTest can't be printed *)
	stringToTestAsString 			:Tc2_System.T_MaxString;
	(* used for placeholder string if expectedString can't be printed *)
	expectedStringAsString 			:Tc2_System.T_MaxString;
	(* contains stringToTest in normalized form *)
	normalizedStringToTest			:WSTRING(Tc2_System.MAX_STRING_LENGTH);
	(* contains expectedString in normalized form *)
	normalizedExpectedString		:WSTRING(Tc2_System.MAX_STRING_LENGTH);
	(* holds characterCount of ``expectedString`` *)
	expectedCharacterCount			:UDINT;
	(* holds characterCount of ``stringToTest`` *)
	stringToTestCharacterCount		:UDINT;
	(* TwinCAT printf with the test message *)
	messageStringBuilder			:Tc2_Utilities.FB_FormatString;
	(* hold stringToCheck before assertion *)
	stringToTestBeforeAssertion		:WSTRING(Tc2_System.MAX_STRING_LENGTH);
	(* hold stringToCheck before assertion *)
	expectedStringBeforeAssertion	:WSTRING(Tc2_System.MAX_STRING_LENGTH);
END_VAR
THIS^.assertorContainer.resetAssertor();

stringToTestBeforeAssertion := stringToTest;
expectedStringBeforeAssertion := expectedString;

CNM_UnicodeUtilities.GetUtf16StringLength(
	utf16StringAddress := ADR(stringToTest),
	characterCount => stringToTestCharacterCount
);
CNM_UnicodeUtilities.GetUtf16StringLength(
	utf16StringAddress := ADR(expectedString),
	characterCount => expectedCharacterCount
);
assertionIsWrong := ((
		stringToTestCharacterCount <> expectedCharacterCount
	) OR (
		CNM_UnicodeUtilities.FindInUtf16String(
			ADR(stringToTest),
			ADR(expectedString),
		) <> 1
	)
);

message := SEL(
	assertionIsWrong,
	'stringToCheck is $'%s$' expected is $'%s$' assertion must be TRUE', 
	'stringToCheck is $'%s$' expected is $'%s$' assertion must be FALSE'
);

Tc2_Utilities.WSTRING_TO_STRING2(ADR(stringToTestAsString), ADR(stringToTest), SIZEOF(stringToTestAsString));
Tc2_Utilities.WSTRING_TO_STRING2(ADR(expectedStringAsString), ADR(expectedString), SIZEOF(expectedStringAsString));

IF (
		Tc2_Standard.WLEN(stringToTest) = TO_UINT(Tc2_System.MAX_STRING_LENGTH)
) THEN
	stringToTestAsString := 'String with Tc2_System.MAX_STRING_LENGTH characters';
END_IF
IF (
		Tc2_Standard.WLEN(expectedString) = TO_UINT(Tc2_System.MAX_STRING_LENGTH)
) THEN
	expectedStringAsString := 'String with Tc2_System.MAX_STRING_LENGTH characters';
END_IF

messageStringBuilder(
	sFormat := message,
	arg1 := THIS^.AnyToArg(stringToTestAsString),
	arg2 := THIS^.AnyToArg(expectedStringAsString)
);
THIS^.assertorContainer.resetAssertor();

THIS^.assertorContainer.assertor.assert.strings.unicode.isEqualTo(
	stringToCheck := stringToTest,
	expected := expectedString,
	ignoreCases := FALSE,
	normalizeStrings := FALSE,
	message			:= ''
);

THIS^.AssertEquals_BOOL(
	Expected 	:= assertionIsWrong,
	Actual 		:= THIS^.assertorContainer.wasAssertionWrong,
	Message 	:= messageStringBuilder.sOut
);

THIS^.AssertEquals_WSTRING(
	Expected 	:= stringToTestBeforeAssertion,
	Actual 		:= stringToTest,
	Message 	:= 'the assertion changed $'stringToTest$''
);

THIS^.AssertEquals_WSTRING(
	Expected 	:= expectedStringBeforeAssertion,
	Actual 		:= expectedString,
	Message 	:= 'the assertion changed $'expectedString$''
);

CNM_UnicodeUtilities.NormalizeUtf16String(
	utf16StringBuffer := ADR(stringToTest),
	bufferSize := Tc2_System.MAX_STRING_LENGTH * 2 + 2,
	normalizedStringBuffer := ADR(normalizedStringToTest),
	normalForm := CNM_UnicodeUtilities.NormalizationForm.NFD
);
CNM_UnicodeUtilities.NormalizeUtf16String(
	utf16StringBuffer := ADR(expectedString),
	bufferSize := Tc2_System.MAX_STRING_LENGTH * 2 + 2,
	normalizedStringBuffer := ADR(normalizedExpectedString),
	normalForm := CNM_UnicodeUtilities.NormalizationForm.NFD
);

CNM_UnicodeUtilities.GetUtf16StringLength(
	utf16StringAddress := ADR(normalizedStringToTest),
	characterCount => stringToTestCharacterCount
);
CNM_UnicodeUtilities.GetUtf16StringLength(
	utf16StringAddress := ADR(normalizedExpectedString),
	characterCount => expectedCharacterCount
);
assertionIsWrong := ((
		stringToTestCharacterCount <> expectedCharacterCount
	) OR (
		CNM_UnicodeUtilities.FindInUtf16String(
			ADR(normalizedStringToTest),
			ADR(normalizedExpectedString),
		) <> 1
	)
);

THIS^.assertorContainer.assertor.assert.strings.unicode.isEqualTo(
	stringToCheck := stringToTest,
	expected := expectedString,
	ignoreCases := FALSE,
	normalizeStrings := TRUE,
	message			:= ''
);

THIS^.AssertEquals_BOOL(
	Expected 	:= assertionIsWrong,
	Actual 		:= THIS^.assertorContainer.wasAssertionWrong,
	Message 	:= messageStringBuilder.sOut
);

THIS^.AssertEquals_WSTRING(
	Expected 	:= stringToTestBeforeAssertion,
	Actual 		:= stringToTest,
	Message 	:= 'the assertion changed $'stringToTest$''
);

THIS^.AssertEquals_WSTRING(
	Expected 	:= expectedStringBeforeAssertion,
	Actual 		:= expectedString,
	Message 	:= 'the assertion changed $'expectedString$''
);
END_METHOD

(*
short summary
==================
This test method tests ``assert.string.unicode.isEqualTo``
method of CNM_AssertionInterfaces library with various inputs

.. <legal notes>

legal notes
=================
| SPDX-FileCopyrightText: © 2022 ekvip automation GmbH <info@ekvip.de>
| SPDX-License-Identifier: Apache-2.0
| For details check: Apache-2.0_

.. _Apache-2.0: https://www.apache.org/licenses/LICENSE-2.0

.. </legal notes>

*)


METHOD testIsEqualToIgnoreCase : BOOL
VAR_INPUT
	(* for the test it's the parameter ``stringToCheck`` *)
	stringToTest  	:WSTRING(Tc2_System.MAX_STRING_LENGTH);
	(* for the test it's the parameter ``searchString`` *)
	expectedString	:WSTRING(Tc2_System.MAX_STRING_LENGTH);
END_VAR
VAR 
	(* just the expectation if the assertion to test must be worng or true *)
	assertionIsWrong				:BOOL;
	(* contains the format string for the test message *)
	message							:Tc2_System.T_MaxString;
	(* contains ´´stringToTest´´ in upper case *)
	upperStringToTest				:WSTRING(Tc2_System.MAX_STRING_LENGTH);
	(* contains ´´expectedString´´ in upper case *)
	upperExpectedString				:WSTRING(Tc2_System.MAX_STRING_LENGTH);
	(* used for placeholder string if stringToTest can't be printed *)
	stringToTestAsString 			:Tc2_System.T_MaxString;
	(* used for placeholder string if expectedString can't be printed *)
	expectedStringAsString 			:Tc2_System.T_MaxString;
	(* contains stringToTest in normalized form *)
	normalizedStringToTest			:WSTRING(Tc2_System.MAX_STRING_LENGTH);
	(* contains expectedString in normalized form *)
	normalizedExpectedString		:WSTRING(Tc2_System.MAX_STRING_LENGTH);
	(* contains stringToTest in normalized form in upper case*)
	normalizedUpperStringToTest		:WSTRING(Tc2_System.MAX_STRING_LENGTH);
	(* contains expectedString in normalized form in upper case*)
	normalizedUpperExpectedString	:WSTRING(Tc2_System.MAX_STRING_LENGTH);
	(* holds characterCount of ``expectedString`` *)
	expectedCharacterCount			:UDINT;
	(* holds characterCount of ``stringToTest`` *)
	stringToTestCharacterCount		:UDINT;
	(* TwinCAT printf with the test message *)
	messageStringBuilder			:Tc2_Utilities.FB_FormatString;
	(* hold stringToCheck before assertion *)
	stringToTestBeforeAssertion		:WSTRING(Tc2_System.MAX_STRING_LENGTH);
	(* hold stringToCheck before assertion *)
	expectedStringBeforeAssertion	:WSTRING(Tc2_System.MAX_STRING_LENGTH);
END_VAR
THIS^.assertorContainer.resetAssertor();

stringToTestBeforeAssertion := stringToTest;
expectedStringBeforeAssertion := expectedString;

upperStringToTest := stringToTest;
upperExpectedString := expectedString;

// both Strings to upper case
CNM_UnicodeUtilities.GetUpperCaseUtf16(ADR(upperStringToTest));
CNM_UnicodeUtilities.GetUpperCaseUtf16(ADR(upperExpectedString));

CNM_UnicodeUtilities.GetUtf16StringLength(
	utf16StringAddress := ADR(upperStringToTest),
	characterCount => stringToTestCharacterCount
);
CNM_UnicodeUtilities.GetUtf16StringLength(
	utf16StringAddress := ADR(upperExpectedString),
	characterCount => expectedCharacterCount
);
assertionIsWrong := ((
		stringToTestCharacterCount <> expectedCharacterCount
	) OR (
		CNM_UnicodeUtilities.FindInUtf16String(
			ADR(upperStringToTest),
			ADR(upperExpectedString),
		) <> 1
	)
);

message := SEL(
	assertionIsWrong,
	'stringToCheck is $'%s$' expected is $'%s$' assertion must be TRUE', 
	'stringToCheck is $'%s$' expected is $'%s$' assertion must be FALSE'
);

Tc2_Utilities.WSTRING_TO_STRING2(ADR(stringToTestAsString), ADR(stringToTest), SIZEOF(stringToTestAsString));
Tc2_Utilities.WSTRING_TO_STRING2(ADR(expectedStringAsString), ADR(expectedString), SIZEOF(expectedStringAsString));

IF (
		Tc2_Standard.WLEN(stringToTest) = TO_UINT(Tc2_System.MAX_STRING_LENGTH)
) THEN
	stringToTestAsString := 'String with Tc2_System.MAX_STRING_LENGTH characters';
END_IF
IF (
		Tc2_Standard.WLEN(expectedString) = TO_UINT(Tc2_System.MAX_STRING_LENGTH)
) THEN
	expectedStringAsString := 'String with Tc2_System.MAX_STRING_LENGTH characters';
END_IF

messageStringBuilder(
	sFormat := message,
	arg1 := THIS^.AnyToArg(stringToTestAsString),
	arg2 := THIS^.AnyToArg(expectedStringAsString)
);
THIS^.assertorContainer.resetAssertor();

THIS^.assertorContainer.assertor.assert.strings.unicode.isEqualTo(
	stringToCheck := stringToTest,
	expected := expectedString,
	ignoreCases := TRUE,
	normalizeStrings := FALSE,
	message			:= ''
);

THIS^.AssertEquals_BOOL(
	Expected 	:= assertionIsWrong,
	Actual 		:= THIS^.assertorContainer.wasAssertionWrong,
	Message 	:= messageStringBuilder.sOut
);

THIS^.AssertEquals_WSTRING(
	Expected 	:= stringToTestBeforeAssertion,
	Actual 		:= stringToTest,
	Message 	:= 'the assertion changed $'stringToTest$''
);

THIS^.AssertEquals_WSTRING(
	Expected 	:= expectedStringBeforeAssertion,
	Actual 		:= expectedString,
	Message 	:= 'the assertion changed $'expectedString$''
);

CNM_UnicodeUtilities.NormalizeUtf16String(
	utf16StringBuffer := ADR(stringToTest),
	bufferSize := Tc2_System.MAX_STRING_LENGTH * 2 + 2,
	normalizedStringBuffer := ADR(normalizedStringToTest),
	normalForm := CNM_UnicodeUtilities.NormalizationForm.NFD
);
CNM_UnicodeUtilities.NormalizeUtf16String(
	utf16StringBuffer := ADR(expectedString),
	bufferSize := Tc2_System.MAX_STRING_LENGTH * 2 + 2,
	normalizedStringBuffer := ADR(normalizedExpectedString),
	normalForm := CNM_UnicodeUtilities.NormalizationForm.NFD
);

normalizedUpperStringToTest := normalizedStringToTest;
normalizedUpperExpectedString := normalizedExpectedString;
CNM_UnicodeUtilities.GetUpperCaseUtf16(ADR(normalizedUpperStringToTest));
CNM_UnicodeUtilities.GetUpperCaseUtf16(ADR(normalizedUpperExpectedString));


CNM_UnicodeUtilities.GetUtf16StringLength(
	utf16StringAddress := ADR(normalizedUpperStringToTest),
	characterCount => stringToTestCharacterCount
);
CNM_UnicodeUtilities.GetUtf16StringLength(
	utf16StringAddress := ADR(normalizedUpperExpectedString),
	characterCount => expectedCharacterCount
);
assertionIsWrong := ((
		stringToTestCharacterCount <> expectedCharacterCount
	) OR (
		CNM_UnicodeUtilities.FindInUtf16String(
			ADR(normalizedUpperStringToTest),
			ADR(normalizedUpperExpectedString),
		) <> 1
	)
);

THIS^.assertorContainer.assertor.assert.strings.unicode.isEqualTo(
	stringToCheck := stringToTest,
	expected := expectedString,
	ignoreCases := TRUE,
	normalizeStrings := TRUE,
	message			:= ''
);

THIS^.AssertEquals_BOOL(
	Expected 	:= assertionIsWrong,
	Actual 		:= THIS^.assertorContainer.wasAssertionWrong,
	Message 	:= messageStringBuilder.sOut
);

THIS^.AssertEquals_WSTRING(
	Expected 	:= stringToTestBeforeAssertion,
	Actual 		:= stringToTest,
	Message 	:= 'the assertion changed $'stringToTest$''
);

THIS^.AssertEquals_WSTRING(
	Expected 	:= expectedStringBeforeAssertion,
	Actual 		:= expectedString,
	Message 	:= 'the assertion changed $'expectedString$''
);
END_METHOD

(*
short summary
==================
This test method tests ``assert.string.unicode.isNotEmpty``
method of CNM_AssertionInterfaces library with various inputs

.. <legal notes>

legal notes
=================
| SPDX-FileCopyrightText: © 2022 ekvip automation GmbH <info@ekvip.de>
| SPDX-License-Identifier: Apache-2.0
| For details check: Apache-2.0_

.. _Apache-2.0: https://www.apache.org/licenses/LICENSE-2.0

.. </legal notes>

*)


METHOD testIsNotEmpty : BOOL
VAR_INPUT
	(* for the test it's the parameter ``stringToCheck`` *)
	stringToTest :WSTRING(Tc2_System.MAX_STRING_LENGTH);
END_VAR
VAR 
	(* just the expectation if the assertion to test must be worng or true *)
	assertionIsWrong				:BOOL;
	(* contains the format string for the test message *)
	message							:Tc2_System.T_MaxString;
	(* used for placeholder string if stringToTest can't be printed *)
	stringToTestAsString 			:Tc2_System.T_MaxString;
	(* holds characterCount of ``stringToTest`` *)
	stringToTestCharacterCount		:UDINT;
	(* TwinCAT printf with the test message *)
	messageStringBuilder			:Tc2_Utilities.FB_FormatString;
	(* hold stringToCheck before assertion *)
	stringToTestBeforeAssertion		:WSTRING(Tc2_System.MAX_STRING_LENGTH);
END_VAR
THIS^.assertorContainer.resetAssertor();

stringToTestBeforeAssertion := stringToTest;

CNM_UnicodeUtilities.GetUtf16StringLength(
	utf16StringAddress := ADR(stringToTest),
	characterCount => stringToTestCharacterCount
);
assertionIsWrong :=  stringToTestCharacterCount = 0;

message := SEL(
	assertionIsWrong,
	'stringToCheck is $'%s$' assertion must be TRUE', 
	'stringToCheck is $'%s$' assertion must be FALSE'
);

Tc2_Utilities.WSTRING_TO_STRING2(ADR(stringToTestAsString), ADR(stringToTest), SIZEOF(stringToTestAsString));

IF (
		Tc2_Standard.WLEN(stringToTest) = TO_UINT(Tc2_System.MAX_STRING_LENGTH)
) THEN
	stringToTestAsString := 'String with Tc2_System.MAX_STRING_LENGTH characters';
END_IF

messageStringBuilder(
	sFormat := message,
	arg1 := THIS^.AnyToArg(stringToTestAsString),
);


THIS^.assertorContainer.assertor.assert.strings.unicode.isNotEmpty(
	stringToCheck := stringToTest,
	message			:= ''
);

THIS^.AssertEquals_BOOL(
	Expected 	:= assertionIsWrong,
	Actual 		:= THIS^.assertorContainer.wasAssertionWrong,
	Message 	:= messageStringBuilder.sOut
);

THIS^.AssertEquals_WSTRING(
	Expected 	:= stringToTestBeforeAssertion,
	Actual 		:= stringToTest,
	Message 	:= 'the assertion changed $'stringToTest$''
);
END_METHOD

(*
short summary
==================
This test method tests ``assert.string.unicode.isNotEqualTo``
method of CNM_AssertionInterfaces library with various inputs

.. <legal notes>

legal notes
=================
| SPDX-FileCopyrightText: © 2022 ekvip automation GmbH <info@ekvip.de>
| SPDX-License-Identifier: Apache-2.0
| For details check: Apache-2.0_

.. _Apache-2.0: https://www.apache.org/licenses/LICENSE-2.0

.. </legal notes>

*)


METHOD testIsNotEqualTo : BOOL
VAR_INPUT
	(* for the test it's the parameter ``stringToCheck`` *)
	stringToTest  	:WSTRING(Tc2_System.MAX_STRING_LENGTH);
	(* for the test it's the parameter ``searchString`` *)
	expectedString	:WSTRING(Tc2_System.MAX_STRING_LENGTH);
END_VAR
VAR 
	(* just the expectation if the assertion to test must be worng or true *)
	assertionIsWrong				:BOOL;
	(* contains the format string for the test message *)
	message							:Tc2_System.T_MaxString;
	(* used for placeholder string if stringToTest can't be printed *)
	stringToTestAsString 			:Tc2_System.T_MaxString;
	(* used for placeholder string if expectedString can't be printed *)
	expectedStringAsString 			:Tc2_System.T_MaxString;
	(* contains stringToTest in normalized form *)
	normalizedStringToTest			:WSTRING(Tc2_System.MAX_STRING_LENGTH);
	(* contains expectedString in normalized form *)
	normalizedExpectedString		:WSTRING(Tc2_System.MAX_STRING_LENGTH);
	(* holds characterCount of ``expectedString`` *)
	expectedCharacterCount			:UDINT;
	(* holds characterCount of ``stringToTest`` *)
	stringToTestCharacterCount		:UDINT;
	(* TwinCAT printf with the test message *)
	messageStringBuilder			:Tc2_Utilities.FB_FormatString;
	(* hold stringToCheck before assertion *)
	stringToTestBeforeAssertion		:WSTRING(Tc2_System.MAX_STRING_LENGTH);
	(* hold stringToCheck before assertion *)
	expectedStringBeforeAssertion	:WSTRING(Tc2_System.MAX_STRING_LENGTH);
END_VAR
THIS^.assertorContainer.resetAssertor();

stringToTestBeforeAssertion := stringToTest;
expectedStringBeforeAssertion := expectedString;

CNM_UnicodeUtilities.GetUtf16StringLength(
	utf16StringAddress := ADR(stringToTest),
	characterCount => stringToTestCharacterCount
);
CNM_UnicodeUtilities.GetUtf16StringLength(
	utf16StringAddress := ADR(expectedString),
	characterCount => expectedCharacterCount
);
assertionIsWrong := ((
		stringToTestCharacterCount = expectedCharacterCount
	) AND (
		CNM_UnicodeUtilities.FindInUtf16String(
			ADR(stringToTest),
			ADR(expectedString),
		) = 1
	)
);

message := SEL(
	assertionIsWrong,
	'stringToCheck is $'%s$' unexpected is $'%s$' assertion must be TRUE', 
	'stringToCheck is $'%s$' unexpected is $'%s$' assertion must be FALSE'
);

Tc2_Utilities.WSTRING_TO_STRING2(ADR(stringToTestAsString), ADR(stringToTest), SIZEOF(stringToTestAsString));
Tc2_Utilities.WSTRING_TO_STRING2(ADR(expectedStringAsString), ADR(expectedString), SIZEOF(expectedStringAsString));

IF (
		Tc2_Standard.WLEN(stringToTest) = TO_UINT(Tc2_System.MAX_STRING_LENGTH)
) THEN
	stringToTestAsString := 'String with Tc2_System.MAX_STRING_LENGTH characters';
END_IF
IF (
		Tc2_Standard.WLEN(expectedString) = TO_UINT(Tc2_System.MAX_STRING_LENGTH)
) THEN
	expectedStringAsString := 'String with Tc2_System.MAX_STRING_LENGTH characters';
END_IF


messageStringBuilder(
	sFormat := message,
	arg1 := THIS^.AnyToArg(stringToTestAsString),
	arg2 := THIS^.AnyToArg(expectedStringAsString)
);


THIS^.assertorContainer.assertor.assert.strings.unicode.isNotEqualTo(
	stringToCheck := stringToTest,
	unexpected := expectedString,
	ignoreCases := FALSE,
	normalizeStrings := FALSE,
	message			:= ''
);

THIS^.AssertEquals_BOOL(
	Expected 	:= assertionIsWrong,
	Actual 		:= THIS^.assertorContainer.wasAssertionWrong,
	Message 	:= messageStringBuilder.sOut
);

THIS^.AssertEquals_WSTRING(
	Expected 	:= stringToTestBeforeAssertion,
	Actual 		:= stringToTest,
	Message 	:= 'the assertion changed $'stringToTest$''
);

THIS^.AssertEquals_WSTRING(
	Expected 	:= expectedStringBeforeAssertion,
	Actual 		:= expectedString,
	Message 	:= 'the assertion changed $'expectedString$''
);

THIS^.assertorContainer.resetAssertor();

CNM_UnicodeUtilities.NormalizeUtf16String(
	utf16StringBuffer := ADR(stringToTest),
	bufferSize := Tc2_System.MAX_STRING_LENGTH * 2 + 2,
	normalizedStringBuffer := ADR(normalizedStringToTest),
	normalForm := CNM_UnicodeUtilities.NormalizationForm.NFD
);
CNM_UnicodeUtilities.NormalizeUtf16String(
	utf16StringBuffer := ADR(expectedString),
	bufferSize := Tc2_System.MAX_STRING_LENGTH * 2 + 2,
	normalizedStringBuffer := ADR(normalizedExpectedString),
	normalForm := CNM_UnicodeUtilities.NormalizationForm.NFD
);

CNM_UnicodeUtilities.GetUtf16StringLength(
	utf16StringAddress := ADR(normalizedStringToTest),
	characterCount => stringToTestCharacterCount
);
CNM_UnicodeUtilities.GetUtf16StringLength(
	utf16StringAddress := ADR(normalizedExpectedString),
	characterCount => expectedCharacterCount
);
assertionIsWrong := ((
		stringToTestCharacterCount = expectedCharacterCount
	) AND (
		CNM_UnicodeUtilities.FindInUtf16String(
			ADR(normalizedStringToTest),
			ADR(normalizedExpectedString),
		) = 1
	)
);

THIS^.assertorContainer.assertor.assert.strings.unicode.isNotEqualTo(
	stringToCheck := stringToTest,
	unexpected := expectedString,
	ignoreCases := FALSE,
	normalizeStrings := TRUE,
	message			:= ''
);

THIS^.AssertEquals_BOOL(
	Expected 	:= assertionIsWrong,
	Actual 		:= THIS^.assertorContainer.wasAssertionWrong,
	Message 	:= messageStringBuilder.sOut
);

THIS^.AssertEquals_WSTRING(
	Expected 	:= stringToTestBeforeAssertion,
	Actual 		:= stringToTest,
	Message 	:= 'the assertion changed $'stringToTest$''
);

THIS^.AssertEquals_WSTRING(
	Expected 	:= expectedStringBeforeAssertion,
	Actual 		:= expectedString,
	Message 	:= 'the assertion changed $'expectedString$''
);
END_METHOD

(*
short summary
==================
This test method tests ``assert.string.unicode.isNotEqualTo``
method of CNM_AssertionInterfaces library with various inputs

.. <legal notes>

legal notes
=================
| SPDX-FileCopyrightText: © 2022 ekvip automation GmbH <info@ekvip.de>
| SPDX-License-Identifier: Apache-2.0
| For details check: Apache-2.0_

.. _Apache-2.0: https://www.apache.org/licenses/LICENSE-2.0

.. </legal notes>

*)


METHOD testIsNotEqualToIgnoreCase : BOOL
VAR_INPUT
	(* for the test it's the parameter ``stringToCheck`` *)
	stringToTest  	:WSTRING(Tc2_System.MAX_STRING_LENGTH);
	(* for the test it's the parameter ``searchString`` *)
	expectedString	:WSTRING(Tc2_System.MAX_STRING_LENGTH);
END_VAR
VAR 
	(* just the expectation if the assertion to test must be worng or true *)
	assertionIsWrong				:BOOL;
	(* contains the format string for the test message *)
	message							:Tc2_System.T_MaxString;
	(* contains ´´stringToTest´´ in upper case *)
	upperStringToTest				:WSTRING(Tc2_System.MAX_STRING_LENGTH);
	(* contains ´´expectedString´´ in upper case *)
	upperExpectedString				:WSTRING(Tc2_System.MAX_STRING_LENGTH);
	(* used for placeholder string if stringToTest can't be printed *)
	stringToTestAsString 			:Tc2_System.T_MaxString;
	(* used for placeholder string if expectedString can't be printed *)
	expectedStringAsString 			:Tc2_System.T_MaxString;
	(* contains stringToTest in normalized form *)
	normalizedStringToTest			:WSTRING(Tc2_System.MAX_STRING_LENGTH);
	(* contains expectedString in normalized form *)
	normalizedExpectedString		:WSTRING(Tc2_System.MAX_STRING_LENGTH);
	(* contains stringToTest in normalized form in upper case*)
	normalizedUpperStringToTest		:WSTRING(Tc2_System.MAX_STRING_LENGTH);
	(* contains expectedString in normalized form in upper case*)
	normalizedUpperExpectedString	:WSTRING(Tc2_System.MAX_STRING_LENGTH);
	(* holds characterCount of ``expectedString`` *)
	expectedCharacterCount			:UDINT;
	(* holds characterCount of ``stringToTest`` *)
	stringToTestCharacterCount		:UDINT;
	(* TwinCAT printf with the test message *)
	messageStringBuilder			:Tc2_Utilities.FB_FormatString;
	(* hold stringToCheck before assertion *)
	stringToTestBeforeAssertion		:WSTRING(Tc2_System.MAX_STRING_LENGTH);
	(* hold stringToCheck before assertion *)
	expectedStringBeforeAssertion	:WSTRING(Tc2_System.MAX_STRING_LENGTH);
END_VAR
THIS^.assertorContainer.resetAssertor();

stringToTestBeforeAssertion := stringToTest;
expectedStringBeforeAssertion := expectedString;

upperStringToTest := stringToTest;
upperExpectedString := expectedString;

// both Strings to upper case
CNM_UnicodeUtilities.GetUpperCaseUtf16(ADR(upperStringToTest));
CNM_UnicodeUtilities.GetUpperCaseUtf16(ADR(upperExpectedString));

CNM_UnicodeUtilities.GetUtf16StringLength(
	utf16StringAddress := ADR(upperStringToTest),
	characterCount => stringToTestCharacterCount
);
CNM_UnicodeUtilities.GetUtf16StringLength(
	utf16StringAddress := ADR(upperExpectedString),
	characterCount => expectedCharacterCount
);
assertionIsWrong := ((
		stringToTestCharacterCount = expectedCharacterCount
	) AND (
		CNM_UnicodeUtilities.FindInUtf16String(
			ADR(upperStringToTest),
			ADR(upperExpectedString),
		) = 1
	)
);

message := SEL(
	assertionIsWrong,
	'stringToCheck is $'%s$' unexpected is $'%s$' assertion must be TRUE', 
	'stringToCheck is $'%s$' unexpected is $'%s$' assertion must be FALSE'
);

Tc2_Utilities.WSTRING_TO_STRING2(ADR(stringToTestAsString), ADR(stringToTest), SIZEOF(stringToTestAsString));
Tc2_Utilities.WSTRING_TO_STRING2(ADR(expectedStringAsString), ADR(expectedString), SIZEOF(expectedStringAsString));

IF (
		Tc2_Standard.WLEN(stringToTest) = TO_UINT(Tc2_System.MAX_STRING_LENGTH)
) THEN
	stringToTestAsString := 'String with Tc2_System.MAX_STRING_LENGTH characters';
END_IF
IF (
		Tc2_Standard.WLEN(expectedString) = TO_UINT(Tc2_System.MAX_STRING_LENGTH)
) THEN
	expectedStringAsString := 'String with Tc2_System.MAX_STRING_LENGTH characters';
END_IF

messageStringBuilder(
	sFormat := message,
	arg1 := THIS^.AnyToArg(stringToTestAsString),
	arg2 := THIS^.AnyToArg(expectedStringAsString)
);
THIS^.assertorContainer.resetAssertor();

THIS^.assertorContainer.assertor.assert.strings.unicode.isNotEqualTo(
	stringToCheck := stringToTest,
	unexpected := expectedString,
	ignoreCases := TRUE,
	normalizeStrings := FALSE,
	message			:= ''
);

THIS^.AssertEquals_BOOL(
	Expected 	:= assertionIsWrong,
	Actual 		:= THIS^.assertorContainer.wasAssertionWrong,
	Message 	:= messageStringBuilder.sOut
);

THIS^.AssertEquals_WSTRING(
	Expected 	:= stringToTestBeforeAssertion,
	Actual 		:= stringToTest,
	Message 	:= 'the assertion changed $'stringToTest$''
);

THIS^.AssertEquals_WSTRING(
	Expected 	:= expectedStringBeforeAssertion,
	Actual 		:= expectedString,
	Message 	:= 'the assertion changed $'expectedString$''
);

CNM_UnicodeUtilities.NormalizeUtf16String(
	utf16StringBuffer := ADR(stringToTest),
	bufferSize := Tc2_System.MAX_STRING_LENGTH * 2 + 2,
	normalizedStringBuffer := ADR(normalizedStringToTest),
	normalForm := CNM_UnicodeUtilities.NormalizationForm.NFD
);
CNM_UnicodeUtilities.NormalizeUtf16String(
	utf16StringBuffer := ADR(expectedString),
	bufferSize := Tc2_System.MAX_STRING_LENGTH * 2 + 2,
	normalizedStringBuffer := ADR(normalizedExpectedString),
	normalForm := CNM_UnicodeUtilities.NormalizationForm.NFD
);

normalizedUpperStringToTest := normalizedStringToTest;
normalizedUpperExpectedString := normalizedExpectedString;
CNM_UnicodeUtilities.GetUpperCaseUtf16(ADR(normalizedUpperStringToTest));
CNM_UnicodeUtilities.GetUpperCaseUtf16(ADR(normalizedUpperExpectedString));


CNM_UnicodeUtilities.GetUtf16StringLength(
	utf16StringAddress := ADR(normalizedUpperStringToTest),
	characterCount => stringToTestCharacterCount
);
CNM_UnicodeUtilities.GetUtf16StringLength(
	utf16StringAddress := ADR(normalizedUpperExpectedString),
	characterCount => expectedCharacterCount
);
assertionIsWrong := ((
		stringToTestCharacterCount = expectedCharacterCount
	) AND (
		CNM_UnicodeUtilities.FindInUtf16String(
			ADR(normalizedUpperStringToTest),
			ADR(normalizedUpperExpectedString),
		) = 1
	)
);

THIS^.assertorContainer.assertor.assert.strings.unicode.isNotEqualTo(
	stringToCheck := stringToTest,
	unexpected := expectedString,
	ignoreCases := TRUE,
	normalizeStrings := TRUE,
	message			:= ''
);

THIS^.AssertEquals_BOOL(
	Expected 	:= assertionIsWrong,
	Actual 		:= THIS^.assertorContainer.wasAssertionWrong,
	Message 	:= messageStringBuilder.sOut
);

THIS^.AssertEquals_WSTRING(
	Expected 	:= stringToTestBeforeAssertion,
	Actual 		:= stringToTest,
	Message 	:= 'the assertion changed $'stringToTest$''
);

THIS^.AssertEquals_WSTRING(
	Expected 	:= expectedStringBeforeAssertion,
	Actual 		:= expectedString,
	Message 	:= 'the assertion changed $'expectedString$''
);
END_METHOD

(*
short summary
==================
This test method tests ``assert.string.unicode.lengthIsBetween``
method of CNM_AssertionInterfaces library with various inputs

.. <legal notes>

legal notes
=================
| SPDX-FileCopyrightText: © 2022 ekvip automation GmbH <info@ekvip.de>
| SPDX-License-Identifier: Apache-2.0
| For details check: Apache-2.0_

.. _Apache-2.0: https://www.apache.org/licenses/LICENSE-2.0

.. </legal notes>

*)


METHOD testLengthIsBetween : BOOL
VAR_INPUT
	(* for the test it's the parameter ``stringToCheck`` *)
	stringToTest			:WSTRING(Tc2_System.MAX_STRING_LENGTH);
	(* for the test it's the parameter ``maxLength`` *)
	maxLength 				:UDINT;
	(* for the test it's the parameter ``minLength`` *)
	minLength 				:UDINT;
	(* UnicodeStringLengthUnit the input is tested for *)
	stringLengthUnit		:CNM_AssertionInterfaces.UnicodeStringLengthUnit;
	(* contains ``stringToTest`` in only ascii charachters for test output *)
	stringToTestPrintable	:Tc2_System.T_MaxString := '';
END_VAR
VAR 
	(* just the expectation if the assertion to test must be worng or true *)
	assertionIsWrong				:BOOL;
	(* contains the format string for the test message *)
	message							:Tc2_System.T_MaxString;
	(* used for placeholder string if stringToTest can't be printed *)
	stringToTestAsString 			:Tc2_System.T_MaxString;
	(* holds string with current ´´stringLengthUnit´´ for the test message*)
	currentStringLengthUnit			:Tc2_System.T_MaxString;
	(* TwinCAT printf with the test message *)
	messageStringBuilder			:Tc2_Utilities.FB_FormatString;
	(* length of current string to check in bytes *)
	stringToTestByteCount			:UDINT;
	(* count of words in current string *)
	stringToTestWordCount			:UDINT;
	(* length of current string to check in characters *)
	stringToTestCodePointCount		:UDINT;
	(* length of ´´stringToCheck´´ *)
	normalizedLength 				:UDINT;
	(* holds the normalized ´´stringToCheck´´ *)
	normalizedStringToTest 			:WSTRING(Tc2_System.MAX_STRING_LENGTH);
	(* width of ´´stringToCheck´´ *)
	stringToTestWidth 				:DINT;
	(* visible characters of ´´stringToCheck´´ *)
	stringToTestVisibleCharacters	:UDINT;
	(*string in UTF32*)
	utf32String						:ARRAY [0..Tc2_System.Global_Variables.MAX_STRING_LENGTH]  OF CNM_UnicodeUtilities.UnicodeCodePoint;
	(* utf32 code point count *)
	utf32CodePointCount 			:UDINT;
	(* bytes in utf8 string *)
	utf8ByteCount 					:UDINT;
	(* hold stringToCheck before assertion *)
	stringToTestBeforeAssertion		:WSTRING(Tc2_System.MAX_STRING_LENGTH);
END_VAR
THIS^.assertorContainer.resetAssertor();

stringToTestBeforeAssertion := stringToTest;

CNM_UnicodeUtilities.GetUtf16StringLength(ADR(stringToTest), wordCount => stringToTestWordCount, characterCount => stringToTestCodePointCount,);
CNM_UnicodeUtilities.GetUtf16StringWidth(ADR(stringToTest), visibleCharacters => stringToTestVisibleCharacters, width => stringToTestWidth);
stringToTestByteCount := stringToTestWordCount * 2;

CNM_UnicodeUtilities.GetCodepointsFromUtf16String(
	utf16StringAddress := ADR(stringToTest),
	utf16StringWordCount := stringToTestWordCount,
	codepointBuffer :=ADR(utf32String),
	bufferSize := SIZEOF(utf32String),
	codePointCount => utf32CodePointCount
);

CNM_UnicodeUtilities.GetUtf8StringFromCodepoints(
	addressOfCodePoints := ADR(utf32String),
	codePointCount := utf32CodePointCount,
	utf8StringBuffer := ADR(stringToTestAsString),
	bufferSize := MAX_STRING_LENGTH + 1,
	utf8StringByteCount => utf8ByteCount
);

IF ( Tc2_Standard.LEN(stringToTestPrintable) <> 0 ) THEN
	stringToTestAsString := stringToTestPrintable;
END_IF


CASE stringLengthUnit OF
	
CNM_AssertionInterfaces.UnicodeStringLengthUnit.BYTES:
	currentStringLengthUnit := 'BYTES';
	
	assertionIsWrong := stringToTestByteCount < minLength OR stringToTestByteCount > maxLength;
	
	message := SEL(
		assertionIsWrong,
		'stringToCheck is $'%s$' with maxLength %u and minLength %u assertion must be TRUE  (%S)', 
		'stringToCheck is $'%s$' with maxLength %u and minLength %u assertion must be FALSE  (%S)'
	);
	
	messageStringBuilder(
		sFormat := message,
		arg1 := THIS^.AnyToArg(stringToTestAsString),
		arg2 := THIS^.AnyToArg(maxLength),
		arg3 := THIS^.AnyToArg(minLength),
		arg4 := THIS^.AnyToArg(currentStringLengthUnit)
	);
	
	THIS^.assertorContainer.assertor.assert.strings.unicode.lengthIsBetween(
		stringToCheck := stringToTest,
		maxLength := maxLength,
		minLength := minLength,
		stringLengthUnit := CNM_AssertionInterfaces.UnicodeStringLengthUnit.BYTES,
		message			:= ''
	);
	
	THIS^.AssertEquals_BOOL(
		Expected 	:= assertionIsWrong,
		Actual 		:= THIS^.assertorContainer.wasAssertionWrong,
		Message 	:= messageStringBuilder.sOut
	);

	THIS^.AssertEquals_WSTRING(
		Expected 	:= stringToTestBeforeAssertion,
		Actual 		:= stringToTest,
		Message 	:= 'the assertion changed $'stringToTest$''
	);

CNM_AssertionInterfaces.UnicodeStringLengthUnit.CHARACTERS:
	currentStringLengthUnit := 'CHARACTERS';
	
	assertionIsWrong := ((
			stringToTestCodePointCount < minLength
		) OR (
			stringToTestCodePointCount > maxLength
		)
	);
	
	message := SEL(
		assertionIsWrong,
		'stringToCheck is $'%s$' with maxLength %u and minLength %u assertion must be TRUE  (%S)', 
		'stringToCheck is $'%s$' with maxLength %u and minLength %u assertion must be FALSE  (%S)'
	);
	
	messageStringBuilder(
		sFormat := message,
		arg1 := THIS^.AnyToArg(stringToTestAsString),
		arg2 := THIS^.AnyToArg(maxLength),
		arg3 := THIS^.AnyToArg(minLength),
		arg4 := THIS^.AnyToArg(currentStringLengthUnit)
	);
	
	THIS^.assertorContainer.assertor.assert.strings.unicode.lengthIsBetween(
		stringToCheck := stringToTest,
		maxLength := maxLength,
		minLength := minLength,
		stringLengthUnit := CNM_AssertionInterfaces.UnicodeStringLengthUnit.CHARACTERS,
		message			:= ''
	);
	
	THIS^.AssertEquals_BOOL(
		Expected 	:= assertionIsWrong,
		Actual 		:= THIS^.assertorContainer.wasAssertionWrong,
		Message 	:= messageStringBuilder.sOut
	);
	
	THIS^.AssertEquals_WSTRING(
		Expected 	:= stringToTestBeforeAssertion,
		Actual 		:= stringToTest,
		Message 	:= 'the assertion changed $'stringToTest$''
	);

CNM_AssertionInterfaces.UnicodeStringLengthUnit.CHARACTERS_NFD:
	currentStringLengthUnit := 'NFD';
	
	CNM_UnicodeUtilities.NormalizeUtf16String(
		utf16StringBuffer := ADR(stringToTest),
		normalForm := CNM_UnicodeUtilities.NormalizationForm.NFD,
		normalizedStringBuffer := ADR(normalizedStringToTest),
		bufferSize := Tc2_System.MAX_STRING_LENGTH * 2 + 2,
		normalizedStringLength => normalizedLength
	);
	CNM_UnicodeUtilities.GetUtf16StringLength(
		utf16StringAddress := ADR(normalizedStringToTest),
		characterCount => stringToTestCodePointCount
	);
		
	assertionIsWrong := ((
			stringToTestCodePointCount < minLength
		) OR (
			stringToTestCodePointCount > maxLength
		)
	);
	
	message := SEL(
		assertionIsWrong,
		'stringToCheck is $'%s$' with maxLength %u and minLength %u assertion must be TRUE  (%S)', 
		'stringToCheck is $'%s$' with maxLength %u and minLength %u assertion must be FALSE  (%S)'
	);
	
	messageStringBuilder(
		sFormat := message,
		arg1 := THIS^.AnyToArg(stringToTestAsString),
		arg2 := THIS^.AnyToArg(maxLength),
		arg3 := THIS^.AnyToArg(minLength),
		arg4 := THIS^.AnyToArg(currentStringLengthUnit)
	);
	
	THIS^.assertorContainer.assertor.assert.strings.unicode.lengthIsBetween(
		stringToCheck := stringToTest,
		maxLength := maxLength,
		minLength := minLength,
		stringLengthUnit := CNM_AssertionInterfaces.UnicodeStringLengthUnit.CHARACTERS_NFD,
		message			:= ''
	);
	
	THIS^.AssertEquals_BOOL(
		Expected 	:= assertionIsWrong,
		Actual 		:= THIS^.assertorContainer.wasAssertionWrong,
		Message 	:= messageStringBuilder.sOut
	);
	
	THIS^.AssertEquals_WSTRING(
		Expected 	:= stringToTestBeforeAssertion,
		Actual 		:= stringToTest,
		Message 	:= 'the assertion changed $'stringToTest$''
	);

CNM_AssertionInterfaces.UnicodeStringLengthUnit.CHARACTERS_NFC:
	currentStringLengthUnit := 'NFC';
	
	CNM_UnicodeUtilities.NormalizeUtf16String(
		utf16StringBuffer := ADR(stringToTest),
		normalForm := CNM_UnicodeUtilities.NormalizationForm.NFC,
		normalizedStringBuffer := ADR(normalizedStringToTest),
		bufferSize := Tc2_System.MAX_STRING_LENGTH * 2 + 2,
		normalizedStringLength => normalizedLength
	);
	CNM_UnicodeUtilities.GetUtf16StringLength(
		utf16StringAddress := ADR(normalizedStringToTest),
		characterCount => stringToTestCodePointCount
	);
		
	assertionIsWrong := ((
			stringToTestCodePointCount < minLength
		) OR (
			stringToTestCodePointCount > maxLength
		)
	);
	
	message := SEL(
		assertionIsWrong,
		'stringToCheck is $'%s$' with maxLength %u and minLength %u assertion must be TRUE  (%S)', 
		'stringToCheck is $'%s$' with maxLength %u and minLength %u assertion must be FALSE  (%S)'
	);
	
	messageStringBuilder(
		sFormat := message,
		arg1 := THIS^.AnyToArg(stringToTestAsString),
		arg2 := THIS^.AnyToArg(maxLength),
		arg3 := THIS^.AnyToArg(minLength),
		arg4 := THIS^.AnyToArg(currentStringLengthUnit)
	);
	
	THIS^.assertorContainer.assertor.assert.strings.unicode.lengthIsBetween(
		stringToCheck := stringToTest,
		maxLength := maxLength,
		minLength := minLength,
		stringLengthUnit := CNM_AssertionInterfaces.UnicodeStringLengthUnit.CHARACTERS_NFC,
		message			:= ''
	);
	
	THIS^.AssertEquals_BOOL(
		Expected 	:= assertionIsWrong,
		Actual 		:= THIS^.assertorContainer.wasAssertionWrong,
		Message 	:= messageStringBuilder.sOut
	);

	THIS^.AssertEquals_WSTRING(
		Expected 	:= stringToTestBeforeAssertion,
		Actual 		:= stringToTest,
		Message 	:= 'the assertion changed $'stringToTest$''
	);

CNM_AssertionInterfaces.UnicodeStringLengthUnit.VISIBLE_CHARACTERS:
	currentStringLengthUnit := 'VISIBLE_CHARACTERS';
	
	assertionIsWrong := ((
			stringToTestVisibleCharacters < minLength
		) OR (
			stringToTestVisibleCharacters > maxLength
		)
	);
	
	message := SEL(
		assertionIsWrong,
		'stringToCheck is $'%s$' with maxLength %u and minLength %u assertion must be TRUE  (%S)', 
		'stringToCheck is $'%s$' with maxLength %u and minLength %u assertion must be FALSE  (%S)'
	);
	
	messageStringBuilder(
		sFormat := message,
		arg1 := THIS^.AnyToArg(stringToTestAsString),
		arg2 := THIS^.AnyToArg(maxLength),
		arg3 := THIS^.AnyToArg(minLength),
		arg4 := THIS^.AnyToArg(currentStringLengthUnit)
	);
	
	THIS^.assertorContainer.assertor.assert.strings.unicode.lengthIsBetween(
		stringToCheck := stringToTest,
		maxLength := maxLength,
		minLength := minLength,
		stringLengthUnit := CNM_AssertionInterfaces.UnicodeStringLengthUnit.VISIBLE_CHARACTERS,
		message			:= ''
	);
	
	THIS^.AssertEquals_BOOL(
		Expected 	:= assertionIsWrong,
		Actual 		:= THIS^.assertorContainer.wasAssertionWrong,
		Message 	:= messageStringBuilder.sOut
	);
	
	THIS^.AssertEquals_WSTRING(
		Expected 	:= stringToTestBeforeAssertion,
		Actual 		:= stringToTest,
		Message 	:= 'the assertion changed $'stringToTest$''
	);
	
CNM_AssertionInterfaces.UnicodeStringLengthUnit.WIDTH:
	currentStringLengthUnit := 'WIDTH';
	
	assertionIsWrong := ((
			TO_UDINT(stringToTestWidth) < minLength
		) OR (
			TO_UDINT(stringToTestWidth) > maxLength
		)
	);
	
	message := SEL(
		assertionIsWrong,
		'stringToCheck is $'%s$' with maxLength %u and minLength %u assertion must be TRUE  (%S)', 
		'stringToCheck is $'%s$' with maxLength %u and minLength %u assertion must be FALSE  (%S)'
	);
	
	messageStringBuilder(
		sFormat := message,
		arg1 := THIS^.AnyToArg(stringToTestAsString),
		arg2 := THIS^.AnyToArg(maxLength),
		arg3 := THIS^.AnyToArg(minLength),
		arg4 := THIS^.AnyToArg(currentStringLengthUnit)
	);
	
	THIS^.assertorContainer.assertor.assert.strings.unicode.lengthIsBetween(
		stringToCheck := stringToTest,
		maxLength := maxLength,
		minLength := minLength,
		stringLengthUnit := CNM_AssertionInterfaces.UnicodeStringLengthUnit.WIDTH,
		message			:= ''
	);
	
	THIS^.AssertEquals_BOOL(
		Expected 	:= assertionIsWrong,
		Actual 		:= THIS^.assertorContainer.wasAssertionWrong,
		Message 	:= messageStringBuilder.sOut
	);

	THIS^.AssertEquals_WSTRING(
		Expected 	:= stringToTestBeforeAssertion,
		Actual 		:= stringToTest,
		Message 	:= 'the assertion changed $'stringToTest$''
	);

END_CASE
END_METHOD

(*
short summary
==================
This test method tests ``assert.string.unicode.lengthIsExact``
method of CNM_AssertionInterfaces library with various inputs

.. <legal notes>

legal notes
=================
| SPDX-FileCopyrightText: © 2022 ekvip automation GmbH <info@ekvip.de>
| SPDX-License-Identifier: Apache-2.0
| For details check: Apache-2.0_

.. _Apache-2.0: https://www.apache.org/licenses/LICENSE-2.0

.. </legal notes>

*)


METHOD testLengthIsExact : BOOL
VAR_INPUT
	(* for the test it's the parameter ``stringToCheck`` *)
	stringToTest 			:WSTRING(Tc2_System.MAX_STRING_LENGTH);
	(* for the test it's the parameter ``expectedLength`` *)
	expectedLength			:UDINT;
	(* UnicodeStringLengthUnit the input is tested for *)
	stringLengthUnit		:CNM_AssertionInterfaces.UnicodeStringLengthUnit;
	(* contains ``stringToTest`` in only ascii charachters for test output *)
	stringToTestPrintable	:Tc2_System.T_MaxString := '';
END_VAR
VAR 
	(* just the expectation if the assertion to test must be worng or true *)
	assertionIsWrong				:BOOL;
	(* contains the format string for the test message *)
	message							:Tc2_System.T_MaxString;
	(* used for placeholder string if stringToTest can't be printed *)
	stringToTestAsString 			:Tc2_System.T_MaxString;
	(* holds string with current ´´stringLengthUnit´´ for the test message*)
	currentStringLengthUnit 		:Tc2_System.T_MaxString;
	(* TwinCAT printf with the test message *)
	messageStringBuilder			:Tc2_Utilities.FB_FormatString;
	(* length of current string to check in bytes *)
	stringToTestByteCount			:UDINT;
	(* count of words in current string *)
	stringToTestWordCount			:UDINT;
	(* length of current string to check in characters *)
	stringToTestCodePointCount		:UDINT;
	(* length of ´´stringToCheck´´ *)
	normalizedLength 				:UDINT;
	(* holds the normalized ´´stringToCheck´´ *)
	normalizedStringToTest 			:WSTRING(Tc2_System.MAX_STRING_LENGTH);
	(* width of ´´stringToCheck´´ *)
	stringToTestWidth 				:DINT;
	(* visible characters of ´´stringToCheck´´ *)
	stringToTestVisibleCharacters	:UDINT := 0;
	(*string in UTF32*)
	utf32String						:ARRAY [0..Tc2_System.Global_Variables.MAX_STRING_LENGTH]  OF CNM_UnicodeUtilities.UnicodeCodePoint;
	(* utf32 code point count *)
	utf32CodePointCount 			:UDINT;
	(* bytes in utf8 string *)
	utf8ByteCount 					:UDINT;
	(* hold stringToCheck before assertion *)
	stringToTestBeforeAssertion		:WSTRING(Tc2_System.MAX_STRING_LENGTH);
END_VAR
THIS^.assertorContainer.resetAssertor();

stringToTestBeforeAssertion := stringToTest;

CNM_UnicodeUtilities.GetUtf16StringLength(ADR(stringToTest), wordCount => stringToTestWordCount, characterCount => stringToTestCodePointCount,);
CNM_UnicodeUtilities.GetUtf16StringWidth(ADR(stringToTest), visibleCharacters => stringToTestVisibleCharacters, width => stringToTestWidth);
stringToTestByteCount := stringToTestWordCount * 2;

CNM_UnicodeUtilities.GetCodepointsFromUtf16String(
	utf16StringAddress := ADR(stringToTest),
	utf16StringWordCount := stringToTestWordCount,
	codepointBuffer :=ADR(utf32String),
	bufferSize := SIZEOF(utf32String),
	codePointCount => utf32CodePointCount
);

CNM_UnicodeUtilities.GetUtf8StringFromCodepoints(
	addressOfCodePoints := ADR(utf32String),
	codePointCount := utf32CodePointCount,
	utf8StringBuffer := ADR(stringToTestAsString),
	bufferSize := MAX_STRING_LENGTH + 1,
	utf8StringByteCount => utf8ByteCount
);

IF ( Tc2_Standard.LEN(stringToTestPrintable) <> 0 ) THEN
	stringToTestAsString := stringToTestPrintable;
END_IF

CASE stringLengthUnit OF
	
CNM_AssertionInterfaces.UnicodeStringLengthUnit.BYTES:
	currentStringLengthUnit := 'BYTES';
	
	assertionIsWrong := stringToTestByteCount <> expectedLength;
	
	message := SEL(
		assertionIsWrong,
		'stringToCheck is $'%s$' with expectedLength %u assertion must be TRUE  (%S)', 
		'stringToCheck is $'%s$' with expectedLength %u assertion must be FALSE  (%S)'
	);
	
	messageStringBuilder(
		sFormat := message,
		arg1 := THIS^.AnyToArg(stringToTestAsString),
		arg2 := THIS^.AnyToArg(expectedLength),
		arg3 := THIS^.AnyToArg(currentStringLengthUnit)
	);
	
	THIS^.assertorContainer.assertor.assert.strings.unicode.lengthIsExact(
		stringToCheck := stringToTest,
		expectedLength := expectedLength,
		stringLengthUnit := CNM_AssertionInterfaces.UnicodeStringLengthUnit.BYTES,
		message			:= ''
	);
	
	THIS^.AssertEquals_BOOL(
		Expected 	:= assertionIsWrong,
		Actual 		:= THIS^.assertorContainer.wasAssertionWrong,
		Message 	:= messageStringBuilder.sOut
	);

	THIS^.AssertEquals_WSTRING(
		Expected 	:= stringToTestBeforeAssertion,
		Actual 		:= stringToTest,
		Message 	:= 'the assertion changed $'stringToTest$''
	);
	
CNM_AssertionInterfaces.UnicodeStringLengthUnit.CHARACTERS:
	currentStringLengthUnit := 'CHARACTERS';
	
	assertionIsWrong := stringToTestCodePointCount <> expectedLength;
	
	message := SEL(
		assertionIsWrong,
		'stringToCheck is $'%s$' with expectedLength %u assertion must be TRUE  (%S)', 
		'stringToCheck is $'%s$' with expectedLength %u assertion must be FALSE  (%S)'
	);
	
	messageStringBuilder(
		sFormat := message,
		arg1 := THIS^.AnyToArg(stringToTestAsString),
		arg2 := THIS^.AnyToArg(expectedLength),
		arg3 := THIS^.AnyToArg(currentStringLengthUnit)
	);
	
	THIS^.assertorContainer.assertor.assert.strings.unicode.lengthIsExact(
		stringToCheck := stringToTest,
		expectedLength := expectedLength,
		stringLengthUnit := CNM_AssertionInterfaces.UnicodeStringLengthUnit.CHARACTERS,
		message			:= ''
	);
	
	THIS^.AssertEquals_BOOL(
		Expected 	:= assertionIsWrong,
		Actual 		:= THIS^.assertorContainer.wasAssertionWrong,
		Message 	:= messageStringBuilder.sOut
	);
	
	THIS^.AssertEquals_WSTRING(
		Expected 	:= stringToTestBeforeAssertion,
		Actual 		:= stringToTest,
		Message 	:= 'the assertion changed $'stringToTest$''
	);
	
CNM_AssertionInterfaces.UnicodeStringLengthUnit.CHARACTERS_NFD:
	currentStringLengthUnit := 'NFD';
	
	CNM_UnicodeUtilities.NormalizeUtf16String(
		utf16StringBuffer := ADR(stringToTest),
		normalForm := CNM_UnicodeUtilities.NormalizationForm.NFD,
		normalizedStringBuffer := ADR(normalizedStringToTest),
		bufferSize := Tc2_System.MAX_STRING_LENGTH * 2 + 2,
		normalizedStringLength => normalizedLength
	);
	CNM_UnicodeUtilities.GetUtf16StringLength(
		utf16StringAddress := ADR(normalizedStringToTest),
		characterCount => stringToTestCodePointCount
	);
		
	assertionIsWrong := stringToTestCodePointCount <> expectedLength;
	
	message := SEL(
		assertionIsWrong,
		'stringToCheck is $'%s$' with expectedLength %u assertion must be TRUE  (%S)', 
		'stringToCheck is $'%s$' with expectedLength %u assertion must be FALSE  (%S)'
	);
	
	messageStringBuilder(
		sFormat := message,
		arg1 := THIS^.AnyToArg(stringToTestAsString),
		arg2 := THIS^.AnyToArg(expectedLength),
		arg3 := THIS^.AnyToArg(currentStringLengthUnit)
	);
	
	THIS^.assertorContainer.assertor.assert.strings.unicode.lengthIsExact(
		stringToCheck := stringToTest,
		expectedLength := expectedLength,
		stringLengthUnit := CNM_AssertionInterfaces.UnicodeStringLengthUnit.CHARACTERS_NFD,
		message			:= ''
	);
	
	THIS^.AssertEquals_BOOL(
		Expected 	:= assertionIsWrong,
		Actual 		:= THIS^.assertorContainer.wasAssertionWrong,
		Message 	:= messageStringBuilder.sOut
	);

	THIS^.AssertEquals_WSTRING(
		Expected 	:= stringToTestBeforeAssertion,
		Actual 		:= stringToTest,
		Message 	:= 'the assertion changed $'stringToTest$''
	);
	
CNM_AssertionInterfaces.UnicodeStringLengthUnit.CHARACTERS_NFC:
	currentStringLengthUnit := 'NFC';
	
	CNM_UnicodeUtilities.NormalizeUtf16String(
		utf16StringBuffer := ADR(stringToTest),
		normalForm := CNM_UnicodeUtilities.NormalizationForm.NFC,
		normalizedStringBuffer := ADR(normalizedStringToTest),
		bufferSize := Tc2_System.MAX_STRING_LENGTH * 2 + 2,
		normalizedStringLength => normalizedLength
	);
	CNM_UnicodeUtilities.GetUtf16StringLength(
		utf16StringAddress := ADR(normalizedStringToTest),
		characterCount => stringToTestCodePointCount
	);
		
	assertionIsWrong := stringToTestCodePointCount <> expectedLength;
	
	message := SEL(
		assertionIsWrong,
		'stringToCheck is $'%s$' with expectedLength %u assertion must be TRUE  (%S)', 
		'stringToCheck is $'%s$' with expectedLength %u assertion must be FALSE  (%S)'
	);
	
	messageStringBuilder(
		sFormat := message,
		arg1 := THIS^.AnyToArg(stringToTestAsString),
		arg2 := THIS^.AnyToArg(expectedLength),
		arg3 := THIS^.AnyToArg(currentStringLengthUnit)
	);
	
